LIN {X 0,Y 528.523,Z 411.8,A -85,B 0,C 180,E1 -4791.18,E2 -4791.18} C_VEL
LIN {X 0,Y 525.787,Z 397.886,A -85,B 0,C 180,E1 -4791.509,E2 -4791.509} C_VEL
LIN {X 0,Y 526.468,Z 375.264,A -85,B 0,C 180,E1 -4794.446,E2 -4794.446} C_VEL
LIN {X 0,Y 526.876,Z 362.602,A -85,B 0,C 180,E1 -4796.116,E2 -4796.116} C_VEL
LIN {X 0,Y 525.642,Z 356.23,A -85,B 0,C 180,E1 -4797.039,E2 -4797.039} C_VEL
LIN {X 0,Y 523.959,Z 348.847,A -85,B 0,C 180,E1 -4798.163,E2 -4798.163} C_VEL
LIN {X 0,Y 523.939,Z 348.847,A -85,B 0,C 180,E1 -4800.854,E2 -4800.854} C_VEL
LIN {X 0,Y 523.93,Z 348.846,A -85,B 0,C 180,E1 -4803.73,E2 -4803.73} C_VEL
LIN {X 0,Y 523.887,Z 348.853,A -85,B 0,C 180,E1 -4806.399,E2 -4806.399} C_VEL
LIN {X 0,Y 523.91,Z 348.844,A -85,B 0,C 180,E1 -4809.086,E2 -4809.086} C_VEL
LIN {X 0,Y 523.909,Z 348.848,A -85,B 0,C 180,E1 -4812.123,E2 -4812.123} C_VEL
LIN {X 0,Y 523.933,Z 348.842,A -85,B 0,C 180,E1 -4815.311,E2 -4815.311} C_VEL
LIN {X 0,Y 523.919,Z 348.849,A -85,B 0,C 180,E1 -4818.695,E2 -4818.695} C_VEL
LIN {X 0,Y 523.903,Z 348.848,A -85,B 0,C 180,E1 -4821.897,E2 -4821.897} C_VEL
LIN {X 0,Y 523.921,Z 348.844,A -85,B 0,C 180,E1 -4824.912,E2 -4824.912} C_VEL
LIN {X 0,Y 523.935,Z 348.841,A -85,B 0,C 180,E1 -4827.68,E2 -4827.68} C_VEL
LIN {X 0,Y 523.952,Z 348.844,A -85,B 0,C 180,E1 -4830.677,E2 -4830.677} C_VEL
LIN {X 0,Y 523.926,Z 348.842,A -85,B 0,C 180,E1 -4833.726,E2 -4833.726} C_VEL
LIN {X 0,Y 523.909,Z 348.852,A -85,B 0,C 180,E1 -4836.27,E2 -4836.27} C_VEL
LIN {X 0,Y 523.945,Z 348.844,A -85,B 0,C 180,E1 -4838.767,E2 -4838.767} C_VEL
LIN {X 0,Y 523.936,Z 348.841,A -85,B 0,C 180,E1 -4841.22,E2 -4841.22} C_VEL
LIN {X 0,Y 523.892,Z 348.846,A -85,B 0,C 180,E1 -4843.638,E2 -4843.638} C_VEL
LIN {X 0,Y 523.925,Z 348.846,A -85,B 0,C 180,E1 -4846.028,E2 -4846.028} C_VEL
LIN {X 0,Y 523.994,Z 348.835,A -85,B 0,C 180,E1 -4849.177,E2 -4849.177} C_VEL
LIN {X 0,Y 523.978,Z 348.84,A -85,B 0,C 180,E1 -4852.292,E2 -4852.292} C_VEL
LIN {X 0,Y 524.067,Z 348.829,A -85,B 0,C 180,E1 -4854.614,E2 -4854.614} C_VEL
LIN {X 0,Y 524.11,Z 348.82,A -85,B 0,C 180,E1 -4857.695,E2 -4857.695} C_VEL
LIN {X 0,Y 524.121,Z 348.823,A -85,B 0,C 180,E1 -4860.769,E2 -4860.769} C_VEL
LIN {X 0,Y 524.031,Z 348.828,A -85,B 0,C 180,E1 -4863.075,E2 -4863.075} C_VEL
LIN {X 0,Y 524.012,Z 348.837,A -85,B 0,C 180,E1 -4866.16,E2 -4866.16} C_VEL
LIN {X 0,Y 523.984,Z 348.836,A -85,B 0,C 180,E1 -4869.263,E2 -4869.263} C_VEL
LIN {X 0,Y 524.002,Z 348.832,A -85,B 0,C 180,E1 -4871.737,E2 -4871.737} C_VEL
LIN {X 0,Y 523.997,Z 348.835,A -85,B 0,C 180,E1 -4875.053,E2 -4875.053} C_VEL
LIN {X 0,Y 523.948,Z 348.841,A -85,B 0,C 180,E1 -4877.97,E2 -4877.97} C_VEL
LIN {X 0,Y 523.975,Z 348.835,A -85,B 0,C 180,E1 -4880.41,E2 -4880.41} C_VEL
LIN {X 0,Y 523.913,Z 348.848,A -85,B 0,C 180,E1 -4882.894,E2 -4882.894} C_VEL
LIN {X 0,Y 523.905,Z 348.838,A -85,B 0,C 180,E1 -4885.422,E2 -4885.422} C_VEL
LIN {X 0,Y 523.917,Z 348.845,A -85,B 0,C 180,E1 -4888.002,E2 -4888.002} C_VEL
LIN {X 0,Y 523.948,Z 348.84,A -85,B 0,C 180,E1 -4890.855,E2 -4890.855} C_VEL
LIN {X 0,Y 523.933,Z 348.843,A -85,B 0,C 180,E1 -4893.73,E2 -4893.73} C_VEL
LIN {X 0,Y 523.892,Z 348.849,A -85,B 0,C 180,E1 -4896.399,E2 -4896.399} C_VEL
LIN {X 0,Y 523.915,Z 348.843,A -85,B 0,C 180,E1 -4899.086,E2 -4899.086} C_VEL
LIN {X 0,Y 523.914,Z 348.848,A -85,B 0,C 180,E1 -4902.123,E2 -4902.123} C_VEL
LIN {X 0,Y 523.944,Z 348.84,A -85,B 0,C 180,E1 -4905.311,E2 -4905.311} C_VEL
LIN {X 0,Y 523.904,Z 348.849,A -85,B 0,C 180,E1 -4906.909,E2 -4906.909} C_VEL
LIN {X 0,Y 523.24,Z 348.929,A -85,B 0,C 180,E1 -4907.551,E2 -4907.551} C_VEL
LIN {X 0,Y 520.398,Z 349.291,A -85,B 0,C 180,E1 -4908.593,E2 -4908.593} C_VEL
LIN {X 0,Y 517.994,Z 349.592,A -85,B 0,C 180,E1 -4909.432,E2 -4909.432} C_VEL
LIN {X 0,Y 516.961,Z 349.719,A -85,B 0,C 180,E1 -4910.08,E2 -4910.08} C_VEL
LIN {X 0,Y 516.877,Z 349.728,A -85,B 0,C 180,E1 -4910.299,E2 -4910.299} C_VEL
LIN {X 0,Y 516.857,Z 349.726,A -85,B 0,C 180,E1 -4913.347,E2 -4913.347} C_VEL
LIN {X 0,Y 516.896,Z 349.753,A -85,B 0,C 180,E1 -4915.084,E2 -4915.084} C_VEL
LIN {X 0,Y 519.011,Z 359.38,A -85,B 0,C 180,E1 -4916.734,E2 -4916.734} C_VEL
LIN {X 0,Y 518.863,Z 369.351,A -85,B 0,C 180,E1 -4918.268,E2 -4918.268} C_VEL
LIN {X 0,Y 521.979,Z 382.993,A -85,B 0,C 180,E1 -4918.604,E2 -4918.604} C_VEL
LIN {X 0,Y 520.819,Z 533.898,A -85,B 0,C 180,E1 -4920.756,E2 -4920.756} C_VEL
LIN {X 0,Y 520.565,Z 549.845,A -85,B 0,C 180,E1 -4921.151,E2 -4921.151} C_VEL
LIN {X 0,Y 520.145,Z 564.573,A -85,B 0,C 180,E1 -4921.675,E2 -4921.675} C_VEL
LIN {X 0,Y 519.695,Z 577.889,A -85,B 0,C 180,E1 -4922.299,E2 -4922.299} C_VEL
LIN {X 0,Y 519.253,Z 591.998,A -85,B 0,C 180,E1 -4923.131,E2 -4923.131} C_VEL
LIN {X 0,Y 518.677,Z 605.217,A -85,B 0,C 180,E1 -4924.088,E2 -4924.088} C_VEL
LIN {X 0,Y 518.211,Z 617.164,A -85,B 0,C 180,E1 -4925.139,E2 -4925.139} C_VEL
LIN {X 0,Y 517.773,Z 627.214,A -85,B 0,C 180,E1 -4926.183,E2 -4926.183} C_VEL
LIN {X 0,Y 517.288,Z 637.933,A -85,B 0,C 180,E1 -4927.499,E2 -4927.499} C_VEL
LIN {X 0,Y 516.945,Z 647.314,A -85,B 0,C 180,E1 -4928.883,E2 -4928.883} C_VEL
LIN {X 0,Y 516.665,Z 655.438,A -85,B 0,C 180,E1 -4930.326,E2 -4930.326} C_VEL
LIN {X 0,Y 516.495,Z 662.099,A -85,B 0,C 180,E1 -4931.762,E2 -4931.762} C_VEL
LIN {X 0,Y 516.351,Z 668.133,A -85,B 0,C 180,E1 -4933.392,E2 -4933.392} C_VEL
LIN {X 0,Y 516.309,Z 672.687,A -85,B 0,C 180,E1 -4935.011,E2 -4935.011} C_VEL
LIN {X 0,Y 516.185,Z 675.904,A -85,B 0,C 180,E1 -4936.617,E2 -4936.617} C_VEL
LIN {X 0,Y 516.231,Z 677.854,A -85,B 0,C 180,E1 -4938.217,E2 -4938.217} C_VEL
LIN {X 0,Y 516.221,Z 678.594,A -85,B 0,C 180,E1 -4939.806,E2 -4939.806} C_VEL
LIN {X 0,Y 516.195,Z 678.184,A -85,B 0,C 180,E1 -4941.387,E2 -4941.387} C_VEL
LIN {X 0,Y 516.284,Z 676.629,A -85,B 0,C 180,E1 -4942.963,E2 -4942.963} C_VEL
LIN {X 0,Y 516.313,Z 673.92,A -85,B 0,C 180,E1 -4944.532,E2 -4944.532} C_VEL
LIN {X 0,Y 516.387,Z 669.998,A -85,B 0,C 180,E1 -4946.098,E2 -4946.098} C_VEL
LIN {X 0,Y 516.37,Z 664.776,A -85,B 0,C 180,E1 -4947.66,E2 -4947.66} C_VEL
LIN {X 0,Y 516.574,Z 658.136,A -85,B 0,C 180,E1 -4949.221,E2 -4949.221} C_VEL
LIN {X 0,Y 516.805,Z 651.008,A -85,B 0,C 180,E1 -4950.584,E2 -4950.584} C_VEL
LIN {X 0,Y 517.127,Z 642.494,A -85,B 0,C 180,E1 -4951.947,E2 -4951.947} C_VEL
LIN {X 0,Y 517.55,Z 632.309,A -85,B 0,C 180,E1 -4953.309,E2 -4953.309} C_VEL
LIN {X 0,Y 517.995,Z 621.915,A -85,B 0,C 180,E1 -4954.474,E2 -4954.474} C_VEL
LIN {X 0,Y 518.569,Z 609.495,A -85,B 0,C 180,E1 -4955.639,E2 -4955.639} C_VEL
LIN {X 0,Y 519.043,Z 597.067,A -85,B 0,C 180,E1 -4956.609,E2 -4956.609} C_VEL
LIN {X 0,Y 519.514,Z 585.147,A -85,B 0,C 180,E1 -4957.384,E2 -4957.384} C_VEL
LIN {X 0,Y 519.995,Z 570.33,A -85,B 0,C 180,E1 -4958.159,E2 -4958.159} C_VEL
LIN {X 0,Y 520.421,Z 555.2,A -85,B 0,C 180,E1 -4958.763,E2 -4958.763} C_VEL
LIN {X 0,Y 520.754,Z 540.07,A -85,B 0,C 180,E1 -4959.198,E2 -4959.198} C_VEL
LIN {X 0,Y 520.967,Z 524.806,A -85,B 0,C 180,E1 -4959.479,E2 -4959.479} C_VEL
LIN {X 0,Y 521.921,Z 382.993,A -85,B 0,C 180,E1 -4961.486,E2 -4961.486} C_VEL
LIN {X 0,Y 518.805,Z 368.955,A -85,B 0,C 180,E1 -4961.848,E2 -4961.848} C_VEL
LIN {X 0,Y 518.989,Z 359.611,A -85,B 0,C 180,E1 -4963.309,E2 -4963.309} C_VEL
LIN {X 0,Y 516.945,Z 349.72,A -85,B 0,C 180,E1 -4965.021,E2 -4965.021} C_VEL
LIN {X 0,Y 516.884,Z 349.724,A -85,B 0,C 180,E1 -4968.224,E2 -4968.224} C_VEL
LIN {X 0,Y 516.91,Z 349.717,A -85,B 0,C 180,E1 -4970.702,E2 -4970.702} C_VEL
LIN {X 0,Y 516.89,Z 349.722,A -85,B 0,C 180,E1 -4974.073,E2 -4974.073} C_VEL
LIN {X 0,Y 516.849,Z 349.725,A -85,B 0,C 180,E1 -4976.662,E2 -4976.662} C_VEL
LIN {X 0,Y 516.891,Z 349.725,A -85,B 0,C 180,E1 -4979.519,E2 -4979.519} C_VEL
LIN {X 0,Y 516.9,Z 349.715,A -85,B 0,C 180,E1 -4982.543,E2 -4982.543} C_VEL
LIN {X 0,Y 516.858,Z 349.729,A -85,B 0,C 180,E1 -4985.327,E2 -4985.327} C_VEL
LIN {X 0,Y 516.88,Z 349.721,A -85,B 0,C 180,E1 -4988.716,E2 -4988.716} C_VEL
LIN {X 0,Y 516.854,Z 349.729,A -85,B 0,C 180,E1 -4991.781,E2 -4991.781} C_VEL
LIN {X 0,Y 516.9,Z 349.718,A -85,B 0,C 180,E1 -4995.007,E2 -4995.007} C_VEL
LIN {X 0,Y 516.891,Z 349.719,A -85,B 0,C 180,E1 -4998.402,E2 -4998.402} C_VEL
LIN {X 0,Y 516.878,Z 349.724,A -85,B 0,C 180,E1 -5001.283,E2 -5001.283} C_VEL
LIN {X 0,Y 516.863,Z 349.722,A -85,B 0,C 180,E1 -5004.671,E2 -5004.671} C_VEL
LIN {X 0,Y 516.898,Z 349.724,A -85,B 0,C 180,E1 -5007.457,E2 -5007.457} C_VEL
LIN {X 0,Y 516.923,Z 349.713,A -85,B 0,C 180,E1 -5010.695,E2 -5010.695} C_VEL
LIN {X 0,Y 516.883,Z 349.711,A -85,B 0,C 180,E1 -5013.818,E2 -5013.818} C_VEL
LIN {X 0,Y 516.862,Z 349.719,A -85,B 0,C 180,E1 -5016.776,E2 -5016.776} C_VEL
LIN {X 0,Y 516.943,Z 349.719,A -85,B 0,C 180,E1 -5019.731,E2 -5019.731} C_VEL
LIN {X 0,Y 516.899,Z 349.713,A -85,B 0,C 180,E1 -5022.595,E2 -5022.595} C_VEL
LIN {X 0,Y 516.939,Z 349.714,A -85,B 0,C 180,E1 -5025.03,E2 -5025.03} C_VEL
LIN {X 0,Y 516.97,Z 349.704,A -85,B 0,C 180,E1 -5028.233,E2 -5028.233} C_VEL
LIN {X 0,Y 516.934,Z 349.718,A -85,B 0,C 180,E1 -5031.399,E2 -5031.399} C_VEL
LIN {X 0,Y 516.99,Z 349.702,A -85,B 0,C 180,E1 -5034.539,E2 -5034.539} C_VEL
LIN {X 0,Y 517.078,Z 349.704,A -85,B 0,C 180,E1 -5037.663,E2 -5037.663} C_VEL
LIN {X 0,Y 517.071,Z 349.697,A -85,B 0,C 180,E1 -5040,E2 -5040} C_VEL
LIN {X 0,Y 517.081,Z 349.693,A -85,B 0,C 180,E1 -5042.337,E2 -5042.337} C_VEL
LIN {X 0,Y 516.978,Z 349.708,A -85,B 0,C 180,E1 -5046.243,E2 -5046.243} C_VEL
LIN {X 0,Y 516.939,Z 349.716,A -85,B 0,C 180,E1 -5049.389,E2 -5049.389} C_VEL
LIN {X 0,Y 516.955,Z 349.714,A -85,B 0,C 180,E1 -5051.806,E2 -5051.806} C_VEL
LIN {X 0,Y 516.941,Z 349.714,A -85,B 0,C 180,E1 -5055.143,E2 -5055.143} C_VEL
LIN {X 0,Y 516.878,Z 349.719,A -85,B 0,C 180,E1 -5058.224,E2 -5058.224} C_VEL
LIN {X 0,Y 516.906,Z 349.716,A -85,B 0,C 180,E1 -5060.701,E2 -5060.701} C_VEL
LIN {X 0,Y 516.886,Z 349.722,A -85,B 0,C 180,E1 -5064.073,E2 -5064.073} C_VEL
LIN {X 0,Y 516.851,Z 349.722,A -85,B 0,C 180,E1 -5066.662,E2 -5066.662} C_VEL
LIN {X 0,Y 516.887,Z 349.727,A -85,B 0,C 180,E1 -5069.518,E2 -5069.518} C_VEL
LIN {X 0,Y 516.896,Z 349.718,A -85,B 0,C 180,E1 -5072.543,E2 -5072.543} C_VEL
LIN {X 0,Y 516.853,Z 349.728,A -85,B 0,C 180,E1 -5075.327,E2 -5075.327} C_VEL
LIN {X 0,Y 516.874,Z 349.719,A -85,B 0,C 180,E1 -5078.716,E2 -5078.716} C_VEL
LIN {X 0,Y 516.85,Z 349.731,A -85,B 0,C 180,E1 -5081.781,E2 -5081.781} C_VEL
LIN {X 0,Y 516.895,Z 349.72,A -85,B 0,C 180,E1 -5085.007,E2 -5085.007} C_VEL
LIN {X 0,Y 516.887,Z 349.721,A -85,B 0,C 180,E1 -5088.402,E2 -5088.402} C_VEL
LIN {X 0,Y 516.873,Z 349.727,A -85,B 0,C 180,E1 -5091.283,E2 -5091.283} C_VEL
LIN {X 0,Y 516.86,Z 349.724,A -85,B 0,C 180,E1 -5094.671,E2 -5094.671} C_VEL
LIN {X 0,Y 516.894,Z 349.726,A -85,B 0,C 180,E1 -5097.457,E2 -5097.457} C_VEL
LIN {X 0,Y 516.92,Z 349.719,A -85,B 0,C 180,E1 -5100.695,E2 -5100.695} C_VEL
LIN {X 0,Y 516.897,Z 349.847,A -85,B 0,C 180,E1 -5101.606,E2 -5101.606} C_VEL
LIN {X 0,Y 519.884,Z 362.48,A -85,B 0,C 180,E1 -5103.506,E2 -5103.506} C_VEL
LIN {X 0,Y 519.893,Z 370.17,A -85,B 0,C 180,E1 -5104.553,E2 -5104.553} C_VEL
LIN {X 0,Y 519.119,Z 391.367,A -85,B 0,C 180,E1 -5107.36,E2 -5107.36} C_VEL
LIN {X 0,Y 518.927,Z 397.801,A -85,B 0,C 180,E1 -5108.203,E2 -5108.203} C_VEL
LIN {X 0,Y 521.926,Z 413.084,A -85,B 0,C 180,E1 -5108.56,E2 -5108.56} C_VEL
LIN {X 0,Y 520.871,Z 563.853,A -85,B 0,C 180,E1 -5110.706,E2 -5110.706} C_VEL
LIN {X 0,Y 520.509,Z 578.962,A -85,B 0,C 180,E1 -5111.066,E2 -5111.066} C_VEL
LIN {X 0,Y 520.139,Z 593.99,A -85,B 0,C 180,E1 -5111.588,E2 -5111.588} C_VEL
LIN {X 0,Y 519.659,Z 607.046,A -85,B 0,C 180,E1 -5112.182,E2 -5112.182} C_VEL
LIN {X 0,Y 519.18,Z 620.988,A -85,B 0,C 180,E1 -5112.978,E2 -5112.978} C_VEL
LIN {X 0,Y 518.647,Z 634.277,A -85,B 0,C 180,E1 -5113.912,E2 -5113.912} C_VEL
LIN {X 0,Y 518.182,Z 645.793,A -85,B 0,C 180,E1 -5114.884,E2 -5114.884} C_VEL
LIN {X 0,Y 517.683,Z 657.488,A -85,B 0,C 180,E1 -5116.056,E2 -5116.056} C_VEL
LIN {X 0,Y 517.304,Z 667.496,A -85,B 0,C 180,E1 -5117.246,E2 -5117.246} C_VEL
LIN {X 0,Y 516.945,Z 677.288,A -85,B 0,C 180,E1 -5118.631,E2 -5118.631} C_VEL
LIN {X 0,Y 516.677,Z 685.457,A -85,B 0,C 180,E1 -5120.013,E2 -5120.013} C_VEL
LIN {X 0,Y 516.54,Z 692.211,A -85,B 0,C 180,E1 -5121.392,E2 -5121.392} C_VEL
LIN {X 0,Y 516.391,Z 698.449,A -85,B 0,C 180,E1 -5122.964,E2 -5122.964} C_VEL
LIN {X 0,Y 516.352,Z 703.276,A -85,B 0,C 180,E1 -5124.533,E2 -5124.533} C_VEL
LIN {X 0,Y 516.307,Z 706.811,A -85,B 0,C 180,E1 -5126.097,E2 -5126.097} C_VEL
LIN {X 0,Y 516.258,Z 709.136,A -85,B 0,C 180,E1 -5127.659,E2 -5127.659} C_VEL
LIN {X 0,Y 516.156,Z 710.303,A -85,B 0,C 180,E1 -5129.22,E2 -5129.22} C_VEL
LIN {X 0,Y 516.156,Z 710.302,A -85,B 0,C 180,E1 -5130.78,E2 -5130.78} C_VEL
LIN {X 0,Y 516.258,Z 709.131,A -85,B 0,C 180,E1 -5132.341,E2 -5132.341} C_VEL
LIN {X 0,Y 516.307,Z 706.806,A -85,B 0,C 180,E1 -5133.903,E2 -5133.903} C_VEL
LIN {X 0,Y 516.351,Z 703.276,A -85,B 0,C 180,E1 -5135.467,E2 -5135.467} C_VEL
LIN {X 0,Y 516.391,Z 698.45,A -85,B 0,C 180,E1 -5137.036,E2 -5137.036} C_VEL
LIN {X 0,Y 516.54,Z 692.202,A -85,B 0,C 180,E1 -5138.607,E2 -5138.607} C_VEL
LIN {X 0,Y 516.757,Z 684.355,A -85,B 0,C 180,E1 -5140.184,E2 -5140.184} C_VEL
LIN {X 0,Y 516.998,Z 676.009,A -85,B 0,C 180,E1 -5141.567,E2 -5141.567} C_VEL
LIN {X 0,Y 517.383,Z 665.957,A -85,B 0,C 180,E1 -5142.952,E2 -5142.952} C_VEL
LIN {X 0,Y 517.747,Z 655.676,A -85,B 0,C 180,E1 -5144.143,E2 -5144.143} C_VEL
LIN {X 0,Y 518.27,Z 643.713,A -85,B 0,C 180,E1 -5145.307,E2 -5145.307} C_VEL
LIN {X 0,Y 518.781,Z 631.145,A -85,B 0,C 180,E1 -5146.326,E2 -5146.326} C_VEL
LIN {X 0,Y 519.326,Z 617.773,A -85,B 0,C 180,E1 -5147.219,E2 -5147.219} C_VEL
LIN {X 0,Y 519.754,Z 605.012,A -85,B 0,C 180,E1 -5147.916,E2 -5147.916} C_VEL
LIN {X 0,Y 520.215,Z 590.051,A -85,B 0,C 180,E1 -5148.562,E2 -5148.562} C_VEL
LIN {X 0,Y 520.547,Z 575.06,A -85,B 0,C 180,E1 -5149.04,E2 -5149.04} C_VEL
LIN {X 0,Y 520.87,Z 559.843,A -85,B 0,C 180,E1 -5149.361,E2 -5149.361} C_VEL
LIN {X 0,Y 521.868,Z 412.692,A -85,B 0,C 180,E1 -5151.448,E2 -5151.448} C_VEL
LIN {X 0,Y 518.907,Z 397.728,A -85,B 0,C 180,E1 -5151.799,E2 -5151.799} C_VEL
LIN {X 0,Y 519.609,Z 376.635,A -85,B 0,C 180,E1 -5154.577,E2 -5154.577} C_VEL
LIN {X 0,Y 520.03,Z 363.985,A -85,B 0,C 180,E1 -5156.27,E2 -5156.27} C_VEL
LIN {X 0,Y 517.499,Z 352.265,A -85,B 0,C 180,E1 -5158.025,E2 -5158.025} C_VEL
LIN {X 0,Y 516.903,Z 349.726,A -85,B 0,C 180,E1 -5158.416,E2 -5158.416} C_VEL
LIN {X 0,Y 516.887,Z 349.724,A -85,B 0,C 180,E1 -5161.11,E2 -5161.11} C_VEL
LIN {X 0,Y 516.885,Z 349.726,A -85,B 0,C 180,E1 -5163.962,E2 -5163.962} C_VEL
LIN {X 0,Y 516.843,Z 349.73,A -85,B 0,C 180,E1 -5166.749,E2 -5166.749} C_VEL
LIN {X 0,Y 516.857,Z 349.723,A -85,B 0,C 180,E1 -5169.724,E2 -5169.724} C_VEL
LIN {X 0,Y 516.883,Z 349.72,A -85,B 0,C 180,E1 -5171.778,E2 -5171.778} C_VEL
LIN {X 0,Y 516.895,Z 349.721,A -85,B 0,C 180,E1 -5175.007,E2 -5175.007} C_VEL
LIN {X 0,Y 516.855,Z 349.731,A -85,B 0,C 180,E1 -5178.406,E2 -5178.406} C_VEL
LIN {X 0,Y 516.873,Z 349.722,A -85,B 0,C 180,E1 -5181.284,E2 -5181.284} C_VEL
LIN {X 0,Y 516.862,Z 349.726,A -85,B 0,C 180,E1 -5184.671,E2 -5184.671} C_VEL
LIN {X 0,Y 516.896,Z 349.717,A -85,B 0,C 180,E1 -5187.457,E2 -5187.457} C_VEL
LIN {X 0,Y 516.919,Z 349.72,A -85,B 0,C 180,E1 -5190.696,E2 -5190.696} C_VEL
LIN {X 0,Y 516.894,Z 349.719,A -85,B 0,C 180,E1 -5193.815,E2 -5193.815} C_VEL
LIN {X 0,Y 516.858,Z 349.726,A -85,B 0,C 180,E1 -5196.776,E2 -5196.776} C_VEL
LIN {X 0,Y 516.938,Z 349.714,A -85,B 0,C 180,E1 -5199.733,E2 -5199.733} C_VEL
LIN {X 0,Y 516.885,Z 349.725,A -85,B 0,C 180,E1 -5202.595,E2 -5202.595} C_VEL
LIN {X 0,Y 516.936,Z 349.715,A -85,B 0,C 180,E1 -5205.03,E2 -5205.03} C_VEL
LIN {X 0,Y 516.968,Z 349.713,A -85,B 0,C 180,E1 -5208.234,E2 -5208.234} C_VEL
LIN {X 0,Y 516.954,Z 349.709,A -85,B 0,C 180,E1 -5211.4,E2 -5211.4} C_VEL
LIN {X 0,Y 517.013,Z 349.709,A -85,B 0,C 180,E1 -5214.54,E2 -5214.54} C_VEL
LIN {X 0,Y 517.081,Z 349.696,A -85,B 0,C 180,E1 -5217.663,E2 -5217.663} C_VEL
LIN {X 0,Y 517.091,Z 349.699,A -85,B 0,C 180,E1 -5220.779,E2 -5220.779} C_VEL
LIN {X 0,Y 516.973,Z 349.707,A -85,B 0,C 180,E1 -5223.118,E2 -5223.118} C_VEL
LIN {X 0,Y 516.977,Z 349.714,A -85,B 0,C 180,E1 -5226.244,E2 -5226.244} C_VEL
LIN {X 0,Y 516.94,Z 349.713,A -85,B 0,C 180,E1 -5229.39,E2 -5229.39} C_VEL
LIN {X 0,Y 516.955,Z 349.71,A -85,B 0,C 180,E1 -5231.807,E2 -5231.807} C_VEL
LIN {X 0,Y 516.948,Z 349.712,A -85,B 0,C 180,E1 -5235.147,E2 -5235.147} C_VEL
LIN {X 0,Y 516.916,Z 349.72,A -85,B 0,C 180,E1 -5238.223,E2 -5238.223} C_VEL
LIN {X 0,Y 516.916,Z 349.718,A -85,B 0,C 180,E1 -5240.702,E2 -5240.702} C_VEL
LIN {X 0,Y 516.889,Z 349.722,A -85,B 0,C 180,E1 -5244.074,E2 -5244.074} C_VEL
LIN {X 0,Y 516.844,Z 349.727,A -85,B 0,C 180,E1 -5246.663,E2 -5246.663} C_VEL
LIN {X 0,Y 516.913,Z 349.715,A -85,B 0,C 180,E1 -5249.524,E2 -5249.524} C_VEL
LIN {X 0,Y 516.898,Z 349.724,A -85,B 0,C 180,E1 -5252.543,E2 -5252.543} C_VEL
LIN {X 0,Y 516.865,Z 349.717,A -85,B 0,C 180,E1 -5255.329,E2 -5255.329} C_VEL
LIN {X 0,Y 516.878,Z 349.723,A -85,B 0,C 180,E1 -5258.717,E2 -5258.717} C_VEL
LIN {X 0,Y 516.888,Z 349.721,A -85,B 0,C 180,E1 -5261.778,E2 -5261.778} C_VEL
LIN {X 0,Y 516.899,Z 349.72,A -85,B 0,C 180,E1 -5265.007,E2 -5265.007} C_VEL
LIN {X 0,Y 516.907,Z 349.723,A -85,B 0,C 180,E1 -5268.4,E2 -5268.4} C_VEL
LIN {X 0,Y 516.877,Z 349.728,A -85,B 0,C 180,E1 -5270.299,E2 -5270.299} C_VEL
LIN {X 0,Y 516.208,Z 349.81,A -85,B 0,C 180,E1 -5270.949,E2 -5270.949} C_VEL
LIN {X 0,Y 513.354,Z 350.164,A -85,B 0,C 180,E1 -5272.005,E2 -5272.005} C_VEL
LIN {X 0,Y 510.938,Z 350.464,A -85,B 0,C 180,E1 -5272.855,E2 -5272.855} C_VEL
LIN {X 0,Y 509.897,Z 350.593,A -85,B 0,C 180,E1 -5273.512,E2 -5273.512} C_VEL
LIN {X 0,Y 509.81,Z 350.604,A -85,B 0,C 180,E1 -5273.734,E2 -5273.734} C_VEL
LIN {X 0,Y 509.891,Z 350.741,A -85,B 0,C 180,E1 -5274.838,E2 -5274.838} C_VEL
LIN {X 0,Y 512.204,Z 361.496,A -85,B 0,C 180,E1 -5276.712,E2 -5276.712} C_VEL
LIN {X 0,Y 512.04,Z 369.598,A -85,B 0,C 180,E1 -5277.963,E2 -5277.963} C_VEL
LIN {X 0,Y 515.38,Z 384.215,A -85,B 0,C 180,E1 -5278.331,E2 -5278.331} C_VEL
LIN {X 0,Y 514.138,Z 534.651,A -85,B 0,C 180,E1 -5280.507,E2 -5280.507} C_VEL
LIN {X 0,Y 513.841,Z 550.586,A -85,B 0,C 180,E1 -5280.912,E2 -5280.912} C_VEL
LIN {X 0,Y 513.405,Z 564.857,A -85,B 0,C 180,E1 -5281.428,E2 -5281.428} C_VEL
LIN {X 0,Y 512.895,Z 579.335,A -85,B 0,C 180,E1 -5282.121,E2 -5282.121} C_VEL
LIN {X 0,Y 512.402,Z 593.563,A -85,B 0,C 180,E1 -5282.989,E2 -5282.989} C_VEL
LIN {X 0,Y 511.803,Z 606.237,A -85,B 0,C 180,E1 -5283.933,E2 -5283.933} C_VEL
LIN {X 0,Y 511.272,Z 618.323,A -85,B 0,C 180,E1 -5285.022,E2 -5285.022} C_VEL
LIN {X 0,Y 510.729,Z 629.847,A -85,B 0,C 180,E1 -5286.265,E2 -5286.265} C_VEL
LIN {X 0,Y 510.284,Z 640.066,A -85,B 0,C 180,E1 -5287.586,E2 -5287.586} C_VEL
LIN {X 0,Y 509.927,Z 649.196,A -85,B 0,C 180,E1 -5289.002,E2 -5289.002} C_VEL
LIN {X 0,Y 509.575,Z 657.01,A -85,B 0,C 180,E1 -5290.461,E2 -5290.461} C_VEL
LIN {X 0,Y 509.412,Z 664.406,A -85,B 0,C 180,E1 -5292.167,E2 -5292.167} C_VEL
LIN {X 0,Y 509.267,Z 669.18,A -85,B 0,C 180,E1 -5293.566,E2 -5293.566} C_VEL
LIN {X 0,Y 509.225,Z 673.127,A -85,B 0,C 180,E1 -5295.04,E2 -5295.04} C_VEL
LIN {X 0,Y 509.1,Z 675.892,A -85,B 0,C 180,E1 -5296.427,E2 -5296.427} C_VEL
LIN {X 0,Y 509.135,Z 677.932,A -85,B 0,C 180,E1 -5298.05,E2 -5298.05} C_VEL
LIN {X 0,Y 509.125,Z 678.785,A -85,B 0,C 180,E1 -5299.662,E2 -5299.662} C_VEL
LIN {X 0,Y 509.104,Z 678.485,A -85,B 0,C 180,E1 -5301.266,E2 -5301.266} C_VEL
LIN {X 0,Y 509.198,Z 677.042,A -85,B 0,C 180,E1 -5302.864,E2 -5302.864} C_VEL
LIN {X 0,Y 509.243,Z 674.44,A -85,B 0,C 180,E1 -5304.456,E2 -5304.456} C_VEL
LIN {X 0,Y 509.311,Z 670.591,A -85,B 0,C 180,E1 -5306.044,E2 -5306.044} C_VEL
LIN {X 0,Y 509.295,Z 665.482,A -85,B 0,C 180,E1 -5307.627,E2 -5307.627} C_VEL
LIN {X 0,Y 509.504,Z 658.974,A -85,B 0,C 180,E1 -5309.21,E2 -5309.21} C_VEL
LIN {X 0,Y 509.755,Z 651.989,A -85,B 0,C 180,E1 -5310.593,E2 -5310.593} C_VEL
LIN {X 0,Y 510.099,Z 643.635,A -85,B 0,C 180,E1 -5311.974,E2 -5311.974} C_VEL
LIN {X 0,Y 510.568,Z 633.63,A -85,B 0,C 180,E1 -5313.354,E2 -5313.354} C_VEL
LIN {X 0,Y 511.017,Z 623.459,A -85,B 0,C 180,E1 -5314.536,E2 -5314.536} C_VEL
LIN {X 0,Y 511.63,Z 611.302,A -85,B 0,C 180,E1 -5315.716,E2 -5315.716} C_VEL
LIN {X 0,Y 512.143,Z 599.208,A -85,B 0,C 180,E1 -5316.698,E2 -5316.698} C_VEL
LIN {X 0,Y 512.705,Z 586.024,A -85,B 0,C 180,E1 -5317.582,E2 -5317.582} C_VEL
LIN {X 0,Y 513.227,Z 571.393,A -85,B 0,C 180,E1 -5318.366,E2 -5318.366} C_VEL
LIN {X 0,Y 513.647,Z 557.269,A -85,B 0,C 180,E1 -5318.954,E2 -5318.954} C_VEL
LIN {X 0,Y 514.083,Z 541.909,A -85,B 0,C 180,E1 -5319.417,E2 -5319.417} C_VEL
LIN {X 0,Y 514.255,Z 527.36,A -85,B 0,C 180,E1 -5319.706,E2 -5319.706} C_VEL
LIN {X 0,Y 515.332,Z 384.044,A -85,B 0,C 180,E1 -5321.762,E2 -5321.762} C_VEL
LIN {X 0,Y 511.944,Z 369.306,A -85,B 0,C 180,E1 -5322.135,E2 -5322.135} C_VEL
LIN {X 0,Y 512.219,Z 362.031,A -85,B 0,C 180,E1 -5323.278,E2 -5323.278} C_VEL
LIN {X 0,Y 510.246,Z 352.192,A -85,B 0,C 180,E1 -5324.967,E2 -5324.967} C_VEL
LIN {X 0,Y 509.908,Z 350.596,A -85,B 0,C 180,E1 -5325.264,E2 -5325.264} C_VEL
LIN {X 0,Y 509.843,Z 350.6,A -85,B 0,C 180,E1 -5328.485,E2 -5328.485} C_VEL
LIN {X 0,Y 509.852,Z 350.597,A -85,B 0,C 180,E1 -5331.002,E2 -5331.002} C_VEL
LIN {X 0,Y 509.824,Z 350.607,A -85,B 0,C 180,E1 -5333.564,E2 -5333.564} C_VEL
LIN {X 0,Y 509.823,Z 350.6,A -85,B 0,C 180,E1 -5336.357,E2 -5336.357} C_VEL
LIN {X 0,Y 509.843,Z 350.598,A -85,B 0,C 180,E1 -5338.846,E2 -5338.846} C_VEL
LIN {X 0,Y 509.824,Z 350.605,A -85,B 0,C 180,E1 -5341.59,E2 -5341.59} C_VEL
LIN {X 0,Y 509.843,Z 350.597,A -85,B 0,C 180,E1 -5344.414,E2 -5344.414} C_VEL
LIN {X 0,Y 509.788,Z 350.607,A -85,B 0,C 180,E1 -5347.344,E2 -5347.344} C_VEL
LIN {X 0,Y 509.818,Z 350.596,A -85,B 0,C 180,E1 -5350.384,E2 -5350.384} C_VEL
LIN {X 0,Y 509.81,Z 350.609,A -85,B 0,C 180,E1 -5353.573,E2 -5353.573} C_VEL
LIN {X 0,Y 509.811,Z 350.596,A -85,B 0,C 180,E1 -5356.427,E2 -5356.427} C_VEL
LIN {X 0,Y 509.816,Z 350.606,A -85,B 0,C 180,E1 -5359.306,E2 -5359.306} C_VEL
LIN {X 0,Y 509.82,Z 350.605,A -85,B 0,C 180,E1 -5361.791,E2 -5361.791} C_VEL
LIN {X 0,Y 509.827,Z 350.599,A -85,B 0,C 180,E1 -5364.621,E2 -5364.621} C_VEL
LIN {X 0,Y 509.864,Z 350.601,A -85,B 0,C 180,E1 -5367.48,E2 -5367.48} C_VEL
LIN {X 0,Y 509.862,Z 350.593,A -85,B 0,C 180,E1 -5370.274,E2 -5370.274} C_VEL
LIN {X 0,Y 509.826,Z 350.589,A -85,B 0,C 180,E1 -5372.94,E2 -5372.94} C_VEL
LIN {X 0,Y 509.838,Z 350.593,A -85,B 0,C 180,E1 -5375.572,E2 -5375.572} C_VEL
LIN {X 0,Y 509.825,Z 350.601,A -85,B 0,C 180,E1 -5378.148,E2 -5378.148} C_VEL
LIN {X 0,Y 509.86,Z 350.594,A -85,B 0,C 180,E1 -5380.681,E2 -5380.681} C_VEL
LIN {X 0,Y 509.868,Z 350.592,A -85,B 0,C 180,E1 -5383.174,E2 -5383.174} C_VEL
LIN {X 0,Y 509.857,Z 350.603,A -85,B 0,C 180,E1 -5385.633,E2 -5385.633} C_VEL
LIN {X 0,Y 509.914,Z 350.582,A -85,B 0,C 180,E1 -5388.874,E2 -5388.874} C_VEL
LIN {X 0,Y 509.88,Z 350.594,A -85,B 0,C 180,E1 -5392.077,E2 -5392.077} C_VEL
LIN {X 0,Y 509.944,Z 350.579,A -85,B 0,C 180,E1 -5394.464,E2 -5394.464} C_VEL
LIN {X 0,Y 510.046,Z 350.58,A -85,B 0,C 180,E1 -5397.631,E2 -5397.631} C_VEL
LIN {X 0,Y 510.04,Z 350.572,A -85,B 0,C 180,E1 -5400,E2 -5400} C_VEL
LIN {X 0,Y 510.051,Z 350.568,A -85,B 0,C 180,E1 -5402.369,E2 -5402.369} C_VEL
LIN {X 0,Y 509.944,Z 350.593,A -85,B 0,C 180,E1 -5405.536,E2 -5405.536} C_VEL
LIN {X 0,Y 509.903,Z 350.587,A -85,B 0,C 180,E1 -5408.72,E2 -5408.72} C_VEL
LIN {X 0,Y 509.906,Z 350.59,A -85,B 0,C 180,E1 -5411.931,E2 -5411.931} C_VEL
LIN {X 0,Y 509.897,Z 350.592,A -85,B 0,C 180,E1 -5415.241,E2 -5415.241} C_VEL
LIN {X 0,Y 509.838,Z 350.595,A -85,B 0,C 180,E1 -5418.484,E2 -5418.484} C_VEL
LIN {X 0,Y 509.848,Z 350.597,A -85,B 0,C 180,E1 -5421.002,E2 -5421.002} C_VEL
LIN {X 0,Y 509.819,Z 350.605,A -85,B 0,C 180,E1 -5423.564,E2 -5423.564} C_VEL
LIN {X 0,Y 509.84,Z 350.596,A -85,B 0,C 180,E1 -5426.361,E2 -5426.361} C_VEL
LIN {X 0,Y 509.839,Z 350.598,A -85,B 0,C 180,E1 -5428.846,E2 -5428.846} C_VEL
LIN {X 0,Y 509.82,Z 350.608,A -85,B 0,C 180,E1 -5431.59,E2 -5431.59} C_VEL
LIN {X 0,Y 509.842,Z 350.598,A -85,B 0,C 180,E1 -5434.414,E2 -5434.414} C_VEL
LIN {X 0,Y 509.783,Z 350.609,A -85,B 0,C 180,E1 -5437.343,E2 -5437.343} C_VEL
LIN {X 0,Y 509.813,Z 350.6,A -85,B 0,C 180,E1 -5440.384,E2 -5440.384} C_VEL
LIN {X 0,Y 509.805,Z 350.61,A -85,B 0,C 180,E1 -5443.573,E2 -5443.573} C_VEL
LIN {X 0,Y 509.807,Z 350.603,A -85,B 0,C 180,E1 -5446.427,E2 -5446.427} C_VEL
LIN {X 0,Y 509.812,Z 350.607,A -85,B 0,C 180,E1 -5449.306,E2 -5449.306} C_VEL
LIN {X 0,Y 509.816,Z 350.607,A -85,B 0,C 180,E1 -5451.791,E2 -5451.791} C_VEL
LIN {X 0,Y 509.824,Z 350.601,A -85,B 0,C 180,E1 -5454.621,E2 -5454.621} C_VEL
LIN {X 0,Y 509.86,Z 350.602,A -85,B 0,C 180,E1 -5457.481,E2 -5457.481} C_VEL
LIN {X 0,Y 509.858,Z 350.6,A -85,B 0,C 180,E1 -5460.274,E2 -5460.274} C_VEL
LIN {X 0,Y 509.869,Z 350.701,A -85,B 0,C 180,E1 -5461.339,E2 -5461.339} C_VEL
LIN {X 0,Y 513.202,Z 365.434,A -85,B 0,C 180,E1 -5463.572,E2 -5463.572} C_VEL
LIN {X 0,Y 512.527,Z 384.409,A -85,B 0,C 180,E1 -5466.139,E2 -5466.139} C_VEL
LIN {X 0,Y 512.1,Z 397.614,A -85,B 0,C 180,E1 -5467.902,E2 -5467.902} C_VEL
LIN {X 0,Y 515.346,Z 414.763,A -85,B 0,C 180,E1 -5468.3,E2 -5468.3} C_VEL
LIN {X 0,Y 514.151,Z 564.432,A -85,B 0,C 180,E1 -5470.46,E2 -5470.46} C_VEL
LIN {X 0,Y 513.763,Z 580.199,A -85,B 0,C 180,E1 -5470.854,E2 -5470.854} C_VEL
LIN {X 0,Y 513.335,Z 595.002,A -85,B 0,C 180,E1 -5471.387,E2 -5471.387} C_VEL
LIN {X 0,Y 512.824,Z 608.809,A -85,B 0,C 180,E1 -5472.04,E2 -5472.04} C_VEL
LIN {X 0,Y 512.27,Z 622.345,A -85,B 0,C 180,E1 -5472.844,E2 -5472.844} C_VEL
LIN {X 0,Y 511.69,Z 636.125,A -85,B 0,C 180,E1 -5473.851,E2 -5473.851} C_VEL
LIN {X 0,Y 511.106,Z 648.597,A -85,B 0,C 180,E1 -5474.957,E2 -5474.957} C_VEL
LIN {X 0,Y 510.586,Z 660.833,A -85,B 0,C 180,E1 -5476.264,E2 -5476.264} C_VEL
LIN {X 0,Y 510.096,Z 671.709,A -85,B 0,C 180,E1 -5477.669,E2 -5477.669} C_VEL
LIN {X 0,Y 509.856,Z 680.772,A -85,B 0,C 180,E1 -5479.074,E2 -5479.074} C_VEL
LIN {X 0,Y 509.52,Z 688.283,A -85,B 0,C 180,E1 -5480.472,E2 -5480.472} C_VEL
LIN {X 0,Y 509.378,Z 695.297,A -85,B 0,C 180,E1 -5482.069,E2 -5482.069} C_VEL
LIN {X 0,Y 509.264,Z 700.811,A -85,B 0,C 180,E1 -5483.661,E2 -5483.661} C_VEL
LIN {X 0,Y 509.158,Z 704.978,A -85,B 0,C 180,E1 -5485.249,E2 -5485.249} C_VEL
LIN {X 0,Y 509.188,Z 707.902,A -85,B 0,C 180,E1 -5486.835,E2 -5486.835} C_VEL
LIN {X 0,Y 509.109,Z 709.643,A -85,B 0,C 180,E1 -5488.418,E2 -5488.418} C_VEL
LIN {X 0,Y 509.062,Z 710.239,A -85,B 0,C 180,E1 -5490,E2 -5490} C_VEL
LIN {X 0,Y 509.109,Z 709.64,A -85,B 0,C 180,E1 -5491.582,E2 -5491.582} C_VEL
LIN {X 0,Y 509.188,Z 707.895,A -85,B 0,C 180,E1 -5493.165,E2 -5493.165} C_VEL
LIN {X 0,Y 509.157,Z 704.972,A -85,B 0,C 180,E1 -5494.751,E2 -5494.751} C_VEL
LIN {X 0,Y 509.237,Z 700.807,A -85,B 0,C 180,E1 -5496.339,E2 -5496.339} C_VEL
LIN {X 0,Y 509.378,Z 695.289,A -85,B 0,C 180,E1 -5497.931,E2 -5497.931} C_VEL
LIN {X 0,Y 509.52,Z 688.263,A -85,B 0,C 180,E1 -5499.527,E2 -5499.527} C_VEL
LIN {X 0,Y 509.851,Z 680.751,A -85,B 0,C 180,E1 -5500.926,E2 -5500.926} C_VEL
LIN {X 0,Y 510.144,Z 671.69,A -85,B 0,C 180,E1 -5502.33,E2 -5502.33} C_VEL
LIN {X 0,Y 510.593,Z 660.805,A -85,B 0,C 180,E1 -5503.735,E2 -5503.735} C_VEL
LIN {X 0,Y 511.111,Z 648.571,A -85,B 0,C 180,E1 -5505.043,E2 -5505.043} C_VEL
LIN {X 0,Y 511.687,Z 636.098,A -85,B 0,C 180,E1 -5506.149,E2 -5506.149} C_VEL
LIN {X 0,Y 512.211,Z 623.828,A -85,B 0,C 180,E1 -5507.055,E2 -5507.055} C_VEL
LIN {X 0,Y 512.751,Z 610.579,A -85,B 0,C 180,E1 -5507.859,E2 -5507.859} C_VEL
LIN {X 0,Y 513.31,Z 596.15,A -85,B 0,C 180,E1 -5508.559,E2 -5508.559} C_VEL
LIN {X 0,Y 513.711,Z 582.109,A -85,B 0,C 180,E1 -5509.082,E2 -5509.082} C_VEL
LIN {X 0,Y 514.058,Z 567.104,A -85,B 0,C 180,E1 -5509.481,E2 -5509.481} C_VEL
LIN {X 0,Y 514.284,Z 545.398,A -85,B 0,C 180,E1 -5509.834,E2 -5509.834} C_VEL
LIN {X 0,Y 515.248,Z 413.666,A -85,B 0,C 180,E1 -5511.719,E2 -5511.719} C_VEL
LIN {X 0,Y 512.054,Z 397.333,A -85,B 0,C 180,E1 -5512.127,E2 -5512.127} C_VEL
LIN {X 0,Y 512.903,Z 374.855,A -85,B 0,C 180,E1 -5515.136,E2 -5515.136} C_VEL
LIN {X 0,Y 513.183,Z 365.393,A -85,B 0,C 180,E1 -5516.429,E2 -5516.429} C_VEL
LIN {X 0,Y 509.854,Z 350.603,A -85,B 0,C 180,E1 -5518.707,E2 -5518.707} C_VEL
LIN {X 0,Y 509.818,Z 350.604,A -85,B 0,C 180,E1 -5521.59,E2 -5521.59} C_VEL
LIN {X 0,Y 509.836,Z 350.606,A -85,B 0,C 180,E1 -5524.415,E2 -5524.415} C_VEL
LIN {X 0,Y 509.793,Z 350.605,A -85,B 0,C 180,E1 -5527.343,E2 -5527.343} C_VEL
LIN {X 0,Y 509.813,Z 350.609,A -85,B 0,C 180,E1 -5530.385,E2 -5530.385} C_VEL
LIN {X 0,Y 509.795,Z 350.605,A -85,B 0,C 180,E1 -5533.059,E2 -5533.059} C_VEL
LIN {X 0,Y 509.82,Z 350.603,A -85,B 0,C 180,E1 -5535.794,E2 -5535.794} C_VEL
LIN {X 0,Y 509.806,Z 350.609,A -85,B 0,C 180,E1 -5538.57,E2 -5538.57} C_VEL
LIN {X 0,Y 509.816,Z 350.602,A -85,B 0,C 180,E1 -5541.659,E2 -5541.659} C_VEL
LIN {X 0,Y 509.825,Z 350.602,A -85,B 0,C 180,E1 -5544.622,E2 -5544.622} C_VEL
LIN {X 0,Y 509.861,Z 350.593,A -85,B 0,C 180,E1 -5547.481,E2 -5547.481} C_VEL
LIN {X 0,Y 509.858,Z 350.593,A -85,B 0,C 180,E1 -5550.274,E2 -5550.274} C_VEL
LIN {X 0,Y 509.871,Z 350.592,A -85,B 0,C 180,E1 -5553.631,E2 -5553.631} C_VEL
LIN {X 0,Y 509.819,Z 350.606,A -85,B 0,C 180,E1 -5556.436,E2 -5556.436} C_VEL
LIN {X 0,Y 509.916,Z 350.59,A -85,B 0,C 180,E1 -5559.845,E2 -5559.845} C_VEL
LIN {X 0,Y 509.847,Z 350.596,A -85,B 0,C 180,E1 -5563.174,E2 -5563.174} C_VEL
LIN {X 0,Y 509.853,Z 350.596,A -85,B 0,C 180,E1 -5565.634,E2 -5565.634} C_VEL
LIN {X 0,Y 509.913,Z 350.591,A -85,B 0,C 180,E1 -5568.875,E2 -5568.875} C_VEL
LIN {X 0,Y 509.91,Z 350.59,A -85,B 0,C 180,E1 -5572.078,E2 -5572.078} C_VEL
LIN {X 0,Y 509.964,Z 350.588,A -85,B 0,C 180,E1 -5574.464,E2 -5574.464} C_VEL
LIN {X 0,Y 510.051,Z 350.572,A -85,B 0,C 180,E1 -5577.631,E2 -5577.631} C_VEL
LIN {X 0,Y 510.041,Z 350.577,A -85,B 0,C 180,E1 -5580.79,E2 -5580.79} C_VEL
LIN {X 0,Y 509.917,Z 350.585,A -85,B 0,C 180,E1 -5583.161,E2 -5583.161} C_VEL
LIN {X 0,Y 509.925,Z 350.594,A -85,B 0,C 180,E1 -5586.331,E2 -5586.331} C_VEL
LIN {X 0,Y 509.88,Z 350.593,A -85,B 0,C 180,E1 -5589.521,E2 -5589.521} C_VEL
LIN {X 0,Y 509.907,Z 350.589,A -85,B 0,C 180,E1 -5591.932,E2 -5591.932} C_VEL
LIN {X 0,Y 509.898,Z 350.59,A -85,B 0,C 180,E1 -5595.242,E2 -5595.242} C_VEL
LIN {X 0,Y 509.86,Z 350.595,A -85,B 0,C 180,E1 -5598.484,E2 -5598.484} C_VEL
LIN {X 0,Y 509.853,Z 350.596,A -85,B 0,C 180,E1 -5601.002,E2 -5601.002} C_VEL
LIN {X 0,Y 509.823,Z 350.599,A -85,B 0,C 180,E1 -5603.564,E2 -5603.564} C_VEL
LIN {X 0,Y 509.819,Z 350.597,A -85,B 0,C 180,E1 -5606.357,E2 -5606.357} C_VEL
LIN {X 0,Y 509.853,Z 350.599,A -85,B 0,C 180,E1 -5608.846,E2 -5608.846} C_VEL
LIN {X 0,Y 509.823,Z 350.595,A -85,B 0,C 180,E1 -5611.59,E2 -5611.59} C_VEL
LIN {X 0,Y 509.84,Z 350.603,A -85,B 0,C 180,E1 -5614.415,E2 -5614.415} C_VEL
LIN {X 0,Y 509.798,Z 350.604,A -85,B 0,C 180,E1 -5617.343,E2 -5617.343} C_VEL
LIN {X 0,Y 509.817,Z 350.604,A -85,B 0,C 180,E1 -5620.385,E2 -5620.385} C_VEL
LIN {X 0,Y 509.799,Z 350.606,A -85,B 0,C 180,E1 -5623.059,E2 -5623.059} C_VEL
LIN {X 0,Y 509.826,Z 350.599,A -85,B 0,C 180,E1 -5625.794,E2 -5625.794} C_VEL
LIN {X 0,Y 509.85,Z 350.604,A -85,B 0,C 180,E1 -5628.574,E2 -5628.574} C_VEL
LIN {X 0,Y 509.854,Z 350.599,A -85,B 0,C 180,E1 -5631.787,E2 -5631.787} C_VEL
LIN {X 0,Y 509.81,Z 350.604,A -85,B 0,C 180,E1 -5633.734,E2 -5633.734} C_VEL
LIN {X 0,Y 509.604,Z 350.993,A -85,B 0,C 180,E1 -5634.169,E2 -5634.169} C_VEL
LIN {X 0,Y 508.77,Z 352.734,A -85,B 0,C 180,E1 -5634.794,E2 -5634.794} C_VEL
LIN {X 0,Y 507.63,Z 355.422,A -85,B 0,C 180,E1 -5635.376,E2 -5635.376} C_VEL
LIN {X 0,Y 506.118,Z 359.963,A -85,B 0,C 180,E1 -5636.126,E2 -5636.126} C_VEL
LIN {X 0,Y 505.373,Z 364.766,A -85,B 0,C 180,E1 -5636.869,E2 -5636.869} C_VEL
LIN {X 0,Y 505.199,Z 369.644,A -85,B 0,C 180,E1 -5637.643,E2 -5637.643} C_VEL
LIN {X 0,Y 508.842,Z 385.728,A -85,B 0,C 180,E1 -5638.057,E2 -5638.057} C_VEL
LIN {X 0,Y 507.469,Z 534.744,A -85,B 0,C 180,E1 -5640.238,E2 -5640.238} C_VEL
LIN {X 0,Y 507.158,Z 550.532,A -85,B 0,C 180,E1 -5640.641,E2 -5640.641} C_VEL
LIN {X 0,Y 506.666,Z 565.309,A -85,B 0,C 180,E1 -5641.183,E2 -5641.183} C_VEL
LIN {X 0,Y 506.174,Z 578.732,A -85,B 0,C 180,E1 -5641.831,E2 -5641.831} C_VEL
LIN {X 0,Y 505.629,Z 592.979,A -85,B 0,C 180,E1 -5642.698,E2 -5642.698} C_VEL
LIN {X 0,Y 504.983,Z 605.91,A -85,B 0,C 180,E1 -5643.665,E2 -5643.665} C_VEL
LIN {X 0,Y 504.438,Z 617.73,A -85,B 0,C 180,E1 -5644.735,E2 -5644.735} C_VEL
LIN {X 0,Y 503.87,Z 628.758,A -85,B 0,C 180,E1 -5645.922,E2 -5645.922} C_VEL
LIN {X 0,Y 503.358,Z 639.106,A -85,B 0,C 180,E1 -5647.249,E2 -5647.249} C_VEL
LIN {X 0,Y 502.922,Z 648.514,A -85,B 0,C 180,E1 -5648.695,E2 -5648.695} C_VEL
LIN {X 0,Y 502.587,Z 656.499,A -85,B 0,C 180,E1 -5650.178,E2 -5650.178} C_VEL
LIN {X 0,Y 502.366,Z 663.202,A -85,B 0,C 180,E1 -5651.695,E2 -5651.695} C_VEL
LIN {X 0,Y 502.205,Z 668.955,A -85,B 0,C 180,E1 -5653.329,E2 -5653.329} C_VEL
LIN {X 0,Y 502.138,Z 673.327,A -85,B 0,C 180,E1 -5654.96,E2 -5654.96} C_VEL
LIN {X 0,Y 502.032,Z 675.854,A -85,B 0,C 180,E1 -5656.232,E2 -5656.232} C_VEL
LIN {X 0,Y 502.037,Z 678.011,A -85,B 0,C 180,E1 -5657.879,E2 -5657.879} C_VEL
LIN {X 0,Y 502.031,Z 678.976,A -85,B 0,C 180,E1 -5659.514,E2 -5659.514} C_VEL
LIN {X 0,Y 502.024,Z 678.787,A -85,B 0,C 180,E1 -5661.142,E2 -5661.142} C_VEL
LIN {X 0,Y 502.108,Z 677.452,A -85,B 0,C 180,E1 -5662.763,E2 -5662.763} C_VEL
LIN {X 0,Y 502.153,Z 674.916,A -85,B 0,C 180,E1 -5664.378,E2 -5664.378} C_VEL
LIN {X 0,Y 502.235,Z 671.175,A -85,B 0,C 180,E1 -5665.988,E2 -5665.988} C_VEL
LIN {X 0,Y 502.222,Z 666.188,A -85,B 0,C 180,E1 -5667.594,E2 -5667.594} C_VEL
LIN {X 0,Y 502.435,Z 659.812,A -85,B 0,C 180,E1 -5669.199,E2 -5669.199} C_VEL
LIN {X 0,Y 502.73,Z 652.967,A -85,B 0,C 180,E1 -5670.601,E2 -5670.601} C_VEL
LIN {X 0,Y 503.072,Z 644.776,A -85,B 0,C 180,E1 -5672.002,E2 -5672.002} C_VEL
LIN {X 0,Y 503.581,Z 634.952,A -85,B 0,C 180,E1 -5673.4,E2 -5673.4} C_VEL
LIN {X 0,Y 504.036,Z 624.975,A -85,B 0,C 180,E1 -5674.599,E2 -5674.599} C_VEL
LIN {X 0,Y 504.688,Z 613.08,A -85,B 0,C 180,E1 -5675.794,E2 -5675.794} C_VEL
LIN {X 0,Y 505.296,Z 599.956,A -85,B 0,C 180,E1 -5676.89,E2 -5676.89} C_VEL
LIN {X 0,Y 505.902,Z 586.861,A -85,B 0,C 180,E1 -5677.785,E2 -5677.785} C_VEL
LIN {X 0,Y 506.458,Z 572.419,A -85,B 0,C 180,E1 -5678.579,E2 -5678.579} C_VEL
LIN {X 0,Y 506.955,Z 557.17,A -85,B 0,C 180,E1 -5679.224,E2 -5679.224} C_VEL
LIN {X 0,Y 507.375,Z 541.365,A -85,B 0,C 180,E1 -5679.701,E2 -5679.701} C_VEL
LIN {X 0,Y 507.619,Z 527.041,A -85,B 0,C 180,E1 -5679.982,E2 -5679.982} C_VEL
LIN {X 0,Y 508.796,Z 385.683,A -85,B 0,C 180,E1 -5682.034,E2 -5682.034} C_VEL
LIN {X 0,Y 505.116,Z 369.466,A -85,B 0,C 180,E1 -5682.454,E2 -5682.454} C_VEL
LIN {X 0,Y 505.291,Z 363.179,A -85,B 0,C 180,E1 -5683.46,E2 -5683.46} C_VEL
LIN {X 0,Y 502.836,Z 351.478,A -85,B 0,C 180,E1 -5685.504,E2 -5685.504} C_VEL
LIN {X 0,Y 502.817,Z 351.476,A -85,B 0,C 180,E1 -5688.752,E2 -5688.752} C_VEL
LIN {X 0,Y 502.787,Z 351.478,A -85,B 0,C 180,E1 -5691.311,E2 -5691.311} C_VEL
LIN {X 0,Y 502.772,Z 351.482,A -85,B 0,C 180,E1 -5693.915,E2 -5693.915} C_VEL
LIN {X 0,Y 502.789,Z 351.476,A -85,B 0,C 180,E1 -5696.571,E2 -5696.571} C_VEL
LIN {X 0,Y 502.815,Z 351.476,A -85,B 0,C 180,E1 -5699.934,E2 -5699.934} C_VEL
LIN {X 0,Y 502.835,Z 351.469,A -85,B 0,C 180,E1 -5703.031,E2 -5703.031} C_VEL
LIN {X 0,Y 502.758,Z 351.48,A -85,B 0,C 180,E1 -5705.953,E2 -5705.953} C_VEL
LIN {X 0,Y 502.79,Z 351.478,A -85,B 0,C 180,E1 -5708.977,E2 -5708.977} C_VEL
LIN {X 0,Y 502.748,Z 351.482,A -85,B 0,C 180,E1 -5712.191,E2 -5712.191} C_VEL
LIN {X 0,Y 502.79,Z 351.478,A -85,B 0,C 180,E1 -5715.47,E2 -5715.47} C_VEL
LIN {X 0,Y 502.799,Z 351.479,A -85,B 0,C 180,E1 -5717.86,E2 -5717.86} C_VEL
LIN {X 0,Y 502.787,Z 351.476,A -85,B 0,C 180,E1 -5721.022,E2 -5721.022} C_VEL
LIN {X 0,Y 502.772,Z 351.479,A -85,B 0,C 180,E1 -5724.17,E2 -5724.17} C_VEL
LIN {X 0,Y 502.807,Z 351.474,A -85,B 0,C 180,E1 -5726.998,E2 -5726.998} C_VEL
LIN {X 0,Y 502.818,Z 351.472,A -85,B 0,C 180,E1 -5730.065,E2 -5730.065} C_VEL
LIN {X 0,Y 502.787,Z 351.466,A -85,B 0,C 180,E1 -5733.429,E2 -5733.429} C_VEL
LIN {X 0,Y 502.771,Z 351.475,A -85,B 0,C 180,E1 -5736.085,E2 -5736.085} C_VEL
LIN {X 0,Y 502.787,Z 351.476,A -85,B 0,C 180,E1 -5738.689,E2 -5738.689} C_VEL
LIN {X 0,Y 502.826,Z 351.475,A -85,B 0,C 180,E1 -5741.248,E2 -5741.248} C_VEL
LIN {X 0,Y 502.852,Z 351.467,A -85,B 0,C 180,E1 -5744.6,E2 -5744.6} C_VEL
LIN {X 0,Y 502.88,Z 351.46,A -85,B 0,C 180,E1 -5748.039,E2 -5748.039} C_VEL
LIN {X 0,Y 502.853,Z 351.469,A -85,B 0,C 180,E1 -5751.156,E2 -5751.156} C_VEL
LIN {X 0,Y 502.874,Z 351.469,A -85,B 0,C 180,E1 -5753.58,E2 -5753.58} C_VEL
LIN {X 0,Y 502.84,Z 351.467,A -85,B 0,C 180,E1 -5756.795,E2 -5756.795} C_VEL
LIN {X 0,Y 502.896,Z 351.462,A -85,B 0,C 180,E1 -5758.398,E2 -5758.398} C_VEL
LIN {X 0,Y 503.009,Z 351.448,A -85,B 0,C 180,E1 -5760,E2 -5760} C_VEL
LIN {X 0,Y 503.02,Z 351.444,A -85,B 0,C 180,E1 -5762.402,E2 -5762.402} C_VEL
LIN {X 0,Y 502.901,Z 351.469,A -85,B 0,C 180,E1 -5765.614,E2 -5765.614} C_VEL
LIN {X 0,Y 502.874,Z 351.465,A -85,B 0,C 180,E1 -5768.033,E2 -5768.033} C_VEL
LIN {X 0,Y 502.878,Z 351.468,A -85,B 0,C 180,E1 -5771.283,E2 -5771.283} C_VEL
LIN {X 0,Y 502.832,Z 351.468,A -85,B 0,C 180,E1 -5774.571,E2 -5774.571} C_VEL
LIN {X 0,Y 502.811,Z 351.472,A -85,B 0,C 180,E1 -5778.109,E2 -5778.109} C_VEL
LIN {X 0,Y 502.831,Z 351.469,A -85,B 0,C 180,E1 -5780.536,E2 -5780.536} C_VEL
LIN {X 0,Y 502.787,Z 351.474,A -85,B 0,C 180,E1 -5783.04,E2 -5783.04} C_VEL
LIN {X 0,Y 502.783,Z 351.482,A -85,B 0,C 180,E1 -5785.678,E2 -5785.678} C_VEL
LIN {X 0,Y 502.775,Z 351.478,A -85,B 0,C 180,E1 -5788.376,E2 -5788.376} C_VEL
LIN {X 0,Y 502.793,Z 351.477,A -85,B 0,C 180,E1 -5791.143,E2 -5791.143} C_VEL
LIN {X 0,Y 502.798,Z 351.479,A -85,B 0,C 180,E1 -5793.994,E2 -5793.994} C_VEL
LIN {X 0,Y 502.737,Z 351.485,A -85,B 0,C 180,E1 -5797.171,E2 -5797.171} C_VEL
LIN {X 0,Y 502.77,Z 351.481,A -85,B 0,C 180,E1 -5800.017,E2 -5800.017} C_VEL
LIN {X 0,Y 502.746,Z 351.484,A -85,B 0,C 180,E1 -5803.234,E2 -5803.234} C_VEL
LIN {X 0,Y 502.779,Z 351.485,A -85,B 0,C 180,E1 -5805.66,E2 -5805.66} C_VEL
LIN {X 0,Y 502.795,Z 351.483,A -85,B 0,C 180,E1 -5807.86,E2 -5807.86} C_VEL
LIN {X 0,Y 502.783,Z 351.48,A -85,B 0,C 180,E1 -5811.022,E2 -5811.022} C_VEL
LIN {X 0,Y 502.768,Z 351.482,A -85,B 0,C 180,E1 -5814.17,E2 -5814.17} C_VEL
LIN {X 0,Y 502.83,Z 351.474,A -85,B 0,C 180,E1 -5816.994,E2 -5816.994} C_VEL
LIN {X 0,Y 502.814,Z 351.479,A -85,B 0,C 180,E1 -5820.065,E2 -5820.065} C_VEL
LIN {X 0,Y 502.859,Z 351.669,A -85,B 0,C 180,E1 -5821.087,E2 -5821.087} C_VEL
LIN {X 0,Y 506.376,Z 366.964,A -85,B 0,C 180,E1 -5823.439,E2 -5823.439} C_VEL
LIN {X 0,Y 505.595,Z 388.601,A -85,B 0,C 180,E1 -5826.397,E2 -5826.397} C_VEL
LIN {X 0,Y 505.238,Z 397.366,A -85,B 0,C 180,E1 -5827.581,E2 -5827.581} C_VEL
LIN {X 0,Y 508.707,Z 416.075,A -85,B 0,C 180,E1 -5828.025,E2 -5828.025} C_VEL
LIN {X 0,Y 507.451,Z 564.218,A -85,B 0,C 180,E1 -5830.192,E2 -5830.192} C_VEL
LIN {X 0,Y 507.02,Z 580.012,A -85,B 0,C 180,E1 -5830.591,E2 -5830.591} C_VEL
LIN {X 0,Y 506.57,Z 595.04,A -85,B 0,C 180,E1 -5831.142,E2 -5831.142} C_VEL
LIN {X 0,Y 506.034,Z 608.576,A -85,B 0,C 180,E1 -5831.791,E2 -5831.791} C_VEL
LIN {X 0,Y 505.439,Z 622.116,A -85,B 0,C 180,E1 -5832.605,E2 -5832.605} C_VEL
LIN {X 0,Y 504.814,Z 635.898,A -85,B 0,C 180,E1 -5833.625,E2 -5833.625} C_VEL
LIN {X 0,Y 504.193,Z 648.372,A -85,B 0,C 180,E1 -5834.746,E2 -5834.746} C_VEL
LIN {X 0,Y 503.684,Z 658.833,A -85,B 0,C 180,E1 -5835.866,E2 -5835.866} C_VEL
LIN {X 0,Y 503.241,Z 668.545,A -85,B 0,C 180,E1 -5837.088,E2 -5837.088} C_VEL
LIN {X 0,Y 502.838,Z 677.688,A -85,B 0,C 180,E1 -5838.447,E2 -5838.447} C_VEL
LIN {X 0,Y 502.608,Z 685.016,A -85,B 0,C 180,E1 -5839.73,E2 -5839.73} C_VEL
LIN {X 0,Y 502.388,Z 691.77,A -85,B 0,C 180,E1 -5841.148,E2 -5841.148} C_VEL
LIN {X 0,Y 502.24,Z 698.011,A -85,B 0,C 180,E1 -5842.765,E2 -5842.765} C_VEL
LIN {X 0,Y 502.181,Z 702.839,A -85,B 0,C 180,E1 -5844.378,E2 -5844.378} C_VEL
LIN {X 0,Y 502.095,Z 706.374,A -85,B 0,C 180,E1 -5845.987,E2 -5845.987} C_VEL
LIN {X 0,Y 502.088,Z 708.7,A -85,B 0,C 180,E1 -5847.593,E2 -5847.593} C_VEL
LIN {X 0,Y 501.986,Z 709.867,A -85,B 0,C 180,E1 -5849.198,E2 -5849.198} C_VEL
LIN {X 0,Y 501.986,Z 709.865,A -85,B 0,C 180,E1 -5850.802,E2 -5850.802} C_VEL
LIN {X 0,Y 502.088,Z 708.692,A -85,B 0,C 180,E1 -5852.407,E2 -5852.407} C_VEL
LIN {X 0,Y 502.095,Z 706.363,A -85,B 0,C 180,E1 -5854.013,E2 -5854.013} C_VEL
LIN {X 0,Y 502.178,Z 702.831,A -85,B 0,C 180,E1 -5855.622,E2 -5855.622} C_VEL
LIN {X 0,Y 502.24,Z 698.002,A -85,B 0,C 180,E1 -5857.235,E2 -5857.235} C_VEL
LIN {X 0,Y 502.388,Z 691.75,A -85,B 0,C 180,E1 -5858.852,E2 -5858.852} C_VEL
LIN {X 0,Y 502.65,Z 683.899,A -85,B 0,C 180,E1 -5860.473,E2 -5860.473} C_VEL
LIN {X 0,Y 502.947,Z 675.891,A -85,B 0,C 180,E1 -5861.842,E2 -5861.842} C_VEL
LIN {X 0,Y 503.393,Z 665.492,A -85,B 0,C 180,E1 -5863.318,E2 -5863.318} C_VEL
LIN {X 0,Y 503.817,Z 655.207,A -85,B 0,C 180,E1 -5864.542,E2 -5864.542} C_VEL
LIN {X 0,Y 504.492,Z 642.817,A -85,B 0,C 180,E1 -5865.776,E2 -5865.776} C_VEL
LIN {X 0,Y 505.086,Z 629.322,A -85,B 0,C 180,E1 -5866.886,E2 -5866.886} C_VEL
LIN {X 0,Y 505.792,Z 615.655,A -85,B 0,C 180,E1 -5867.8,E2 -5867.8} C_VEL
LIN {X 0,Y 506.327,Z 601.498,A -85,B 0,C 180,E1 -5868.565,E2 -5868.565} C_VEL
LIN {X 0,Y 506.842,Z 586.181,A -85,B 0,C 180,E1 -5869.202,E2 -5869.202} C_VEL
LIN {X 0,Y 507.286,Z 570.955,A -85,B 0,C 180,E1 -5869.657,E2 -5869.657} C_VEL
LIN {X 0,Y 507.517,Z 554.938,A -85,B 0,C 180,E1 -5869.964,E2 -5869.964} C_VEL
LIN {X 0,Y 508.713,Z 415.844,A -85,B 0,C 180,E1 -5871.977,E2 -5871.977} C_VEL
LIN {X 0,Y 505.232,Z 397.119,A -85,B 0,C 180,E1 -5872.442,E2 -5872.442} C_VEL
LIN {X 0,Y 506.108,Z 375.669,A -85,B 0,C 180,E1 -5875.361,E2 -5875.361} C_VEL
LIN {X 0,Y 506.365,Z 367.043,A -85,B 0,C 180,E1 -5876.561,E2 -5876.561} C_VEL
LIN {X 0,Y 503.107,Z 352.698,A -85,B 0,C 180,E1 -5878.812,E2 -5878.812} C_VEL
LIN {X 0,Y 502.811,Z 351.478,A -85,B 0,C 180,E1 -5879.03,E2 -5879.03} C_VEL
LIN {X 0,Y 502.782,Z 351.484,A -85,B 0,C 180,E1 -5882.085,E2 -5882.085} C_VEL
LIN {X 0,Y 502.792,Z 351.48,A -85,B 0,C 180,E1 -5884.966,E2 -5884.966} C_VEL
LIN {X 0,Y 502.763,Z 351.482,A -85,B 0,C 180,E1 -5888.482,E2 -5888.482} C_VEL
LIN {X 0,Y 502.771,Z 351.478,A -85,B 0,C 180,E1 -5891.071,E2 -5891.071} C_VEL
LIN {X 0,Y 502.752,Z 351.481,A -85,B 0,C 180,E1 -5893.372,E2 -5893.372} C_VEL
LIN {X 0,Y 502.777,Z 351.479,A -85,B 0,C 180,E1 -5895.66,E2 -5895.66} C_VEL
LIN {X 0,Y 502.764,Z 351.481,A -85,B 0,C 180,E1 -5899.013,E2 -5899.013} C_VEL
LIN {X 0,Y 502.764,Z 351.484,A -85,B 0,C 180,E1 -5902.044,E2 -5902.044} C_VEL
LIN {X 0,Y 502.796,Z 351.475,A -85,B 0,C 180,E1 -5905.034,E2 -5905.034} C_VEL
LIN {X 0,Y 502.783,Z 351.478,A -85,B 0,C 180,E1 -5907.916,E2 -5907.916} C_VEL
LIN {X 0,Y 502.812,Z 351.477,A -85,B 0,C 180,E1 -5910.712,E2 -5910.712} C_VEL
LIN {X 0,Y 502.822,Z 351.47,A -85,B 0,C 180,E1 -5913.449,E2 -5913.449} C_VEL
LIN {X 0,Y 502.768,Z 351.483,A -85,B 0,C 180,E1 -5916.085,E2 -5916.085} C_VEL
LIN {X 0,Y 502.782,Z 351.482,A -85,B 0,C 180,E1 -5918.689,E2 -5918.689} C_VEL
LIN {X 0,Y 502.812,Z 351.473,A -85,B 0,C 180,E1 -5921.248,E2 -5921.248} C_VEL
LIN {X 0,Y 502.838,Z 351.475,A -85,B 0,C 180,E1 -5924.664,E2 -5924.664} C_VEL
LIN {X 0,Y 502.878,Z 351.466,A -85,B 0,C 180,E1 -5928.04,E2 -5928.04} C_VEL
LIN {X 0,Y 502.863,Z 351.465,A -85,B 0,C 180,E1 -5931.157,E2 -5931.157} C_VEL
LIN {X 0,Y 502.918,Z 351.467,A -85,B 0,C 180,E1 -5934.387,E2 -5934.387} C_VEL
LIN {X 0,Y 503.02,Z 351.447,A -85,B 0,C 180,E1 -5937.598,E2 -5937.598} C_VEL
LIN {X 0,Y 502.992,Z 351.455,A -85,B 0,C 180,E1 -5940.801,E2 -5940.801} C_VEL
LIN {X 0,Y 503.019,Z 351.454,A -85,B 0,C 180,E1 -5942.403,E2 -5942.403} C_VEL
LIN {X 0,Y 502.919,Z 351.46,A -85,B 0,C 180,E1 -5945.614,E2 -5945.614} C_VEL
LIN {X 0,Y 502.863,Z 351.471,A -85,B 0,C 180,E1 -5948.844,E2 -5948.844} C_VEL
LIN {X 0,Y 502.848,Z 351.47,A -85,B 0,C 180,E1 -5952.102,E2 -5952.102} C_VEL
LIN {X 0,Y 502.852,Z 351.467,A -85,B 0,C 180,E1 -5955.4,E2 -5955.4} C_VEL
LIN {X 0,Y 502.826,Z 351.466,A -85,B 0,C 180,E1 -5958.752,E2 -5958.752} C_VEL
LIN {X 0,Y 502.786,Z 351.475,A -85,B 0,C 180,E1 -5961.312,E2 -5961.312} C_VEL
LIN {X 0,Y 502.772,Z 351.479,A -85,B 0,C 180,E1 -5963.915,E2 -5963.915} C_VEL
LIN {X 0,Y 502.786,Z 351.476,A -85,B 0,C 180,E1 -5966.571,E2 -5966.571} C_VEL
LIN {X 0,Y 502.816,Z 351.472,A -85,B 0,C 180,E1 -5969.289,E2 -5969.289} C_VEL
LIN {X 0,Y 502.786,Z 351.475,A -85,B 0,C 180,E1 -5972.085,E2 -5972.085} C_VEL
LIN {X 0,Y 502.796,Z 351.472,A -85,B 0,C 180,E1 -5974.967,E2 -5974.967} C_VEL
LIN {X 0,Y 502.768,Z 351.483,A -85,B 0,C 180,E1 -5978.482,E2 -5978.482} C_VEL
LIN {X 0,Y 502.775,Z 351.48,A -85,B 0,C 180,E1 -5981.071,E2 -5981.071} C_VEL
LIN {X 0,Y 502.757,Z 351.482,A -85,B 0,C 180,E1 -5983.372,E2 -5983.372} C_VEL
LIN {X 0,Y 502.783,Z 351.476,A -85,B 0,C 180,E1 -5985.66,E2 -5985.66} C_VEL
LIN {X 0,Y 502.8,Z 351.48,A -85,B 0,C 180,E1 -5988.932,E2 -5988.932} C_VEL
LIN {X 0,Y 502.794,Z 351.48,A -85,B 0,C 180,E1 -5992.046,E2 -5992.046} C_VEL
LIN {X 0,Y 502.809,Z 351.555,A -85,B 0,C 180,E1 -5994.545,E2 -5994.545} C_VEL
LIN {X 0,Y 505.317,Z 362.901,A -85,B 0,C 180,E1 -5996.563,E2 -5996.563} C_VEL
LIN {X 0,Y 505.373,Z 364.766,A -85,B 0,C 180,E1 -5996.869,E2 -5996.869} C_VEL
LIN {X 0,Y 505.19,Z 367.437,A -85,B 0,C 180,E1 -5997.184,E2 -5997.184} C_VEL
LIN {X 0,Y 504.555,Z 372.52,A -85,B 0,C 180,E1 -5997.504,E2 -5997.504} C_VEL
LIN {X 0,Y 503.729,Z 378.198,A -85,B 0,C 180,E1 -5997.682,E2 -5997.682} C_VEL
LIN {X 0,Y 502.215,Z 388.62,A -85,B 0,C 180,E1 -5997.788,E2 -5997.788} C_VEL
LIN {X 0,Y 502.192,Z 394.914,A -85,B 0,C 180,E1 -5997.884,E2 -5997.884} C_VEL
LIN {X 0,Y 500.818,Z 534.85,A -85,B 0,C 180,E1 -5999.961,E2 -5999.961} C_VEL
LIN {X 0,Y 500.438,Z 550.757,A -85,B 0,C 180,E1 -6000.371,E2 -6000.371} C_VEL
LIN {X 0,Y 499.941,Z 565.942,A -85,B 0,C 180,E1 -6000.939,E2 -6000.939} C_VEL
LIN {X 0,Y 499.382,Z 580.141,A -85,B 0,C 180,E1 -6001.642,E2 -6001.642} C_VEL
LIN {X 0,Y 498.822,Z 593.99,A -85,B 0,C 180,E1 -6002.51,E2 -6002.51} C_VEL
LIN {X 0,Y 498.103,Z 606.913,A -85,B 0,C 180,E1 -6003.499,E2 -6003.499} C_VEL
LIN {X 0,Y 497.51,Z 619.16,A -85,B 0,C 180,E1 -6004.638,E2 -6004.638} C_VEL
LIN {X 0,Y 496.813,Z 631.317,A -85,B 0,C 180,E1 -6006.002,E2 -6006.002} C_VEL
LIN {X 0,Y 496.344,Z 640.555,A -85,B 0,C 180,E1 -6007.238,E2 -6007.238} C_VEL
LIN {X 0,Y 495.873,Z 650.376,A -85,B 0,C 180,E1 -6008.813,E2 -6008.813} C_VEL
LIN {X 0,Y 495.441,Z 659.03,A -85,B 0,C 180,E1 -6010.527,E2 -6010.527} C_VEL
LIN {X 0,Y 495.289,Z 664.833,A -85,B 0,C 180,E1 -6011.938,E2 -6011.938} C_VEL
LIN {X 0,Y 495.134,Z 670.002,A -85,B 0,C 180,E1 -6013.508,E2 -6013.508} C_VEL
LIN {X 0,Y 495.049,Z 674.213,A -85,B 0,C 180,E1 -6015.195,E2 -6015.195} C_VEL
LIN {X 0,Y 494.93,Z 677.106,A -85,B 0,C 180,E1 -6016.868,E2 -6016.868} C_VEL
LIN {X 0,Y 494.992,Z 678.773,A -85,B 0,C 180,E1 -6018.535,E2 -6018.535} C_VEL
LIN {X 0,Y 494.917,Z 679.271,A -85,B 0,C 180,E1 -6020.189,E2 -6020.189} C_VEL
LIN {X 0,Y 494.945,Z 678.607,A -85,B 0,C 180,E1 -6021.837,E2 -6021.837} C_VEL
LIN {X 0,Y 495.068,Z 676.607,A -85,B 0,C 180,E1 -6023.581,E2 -6023.581} C_VEL
LIN {X 0,Y 495.007,Z 673.732,A -85,B 0,C 180,E1 -6025.113,E2 -6025.113} C_VEL
LIN {X 0,Y 495.204,Z 669.484,A -85,B 0,C 180,E1 -6026.746,E2 -6026.746} C_VEL
LIN {X 0,Y 495.223,Z 663.955,A -85,B 0,C 180,E1 -6028.374,E2 -6028.374} C_VEL
LIN {X 0,Y 495.61,Z 656.949,A -85,B 0,C 180,E1 -6030,E2 -6030} C_VEL
LIN {X 0,Y 495.894,Z 649.508,A -85,B 0,C 180,E1 -6031.421,E2 -6031.421} C_VEL
LIN {X 0,Y 496.373,Z 640.586,A -85,B 0,C 180,E1 -6032.841,E2 -6032.841} C_VEL
LIN {X 0,Y 496.901,Z 629.875,A -85,B 0,C 180,E1 -6034.258,E2 -6034.258} C_VEL
LIN {X 0,Y 497.495,Z 618.916,A -85,B 0,C 180,E1 -6035.472,E2 -6035.472} C_VEL
LIN {X 0,Y 498.159,Z 606.922,A -85,B 0,C 180,E1 -6036.582,E2 -6036.582} C_VEL
LIN {X 0,Y 498.787,Z 593.798,A -85,B 0,C 180,E1 -6037.591,E2 -6037.591} C_VEL
LIN {X 0,Y 499.495,Z 579.164,A -85,B 0,C 180,E1 -6038.496,E2 -6038.496} C_VEL
LIN {X 0,Y 500.059,Z 564.683,A -85,B 0,C 180,E1 -6039.199,E2 -6039.199} C_VEL
LIN {X 0,Y 500.538,Z 550.372,A -85,B 0,C 180,E1 -6039.725,E2 -6039.725} C_VEL
LIN {X 0,Y 500.783,Z 535.311,A -85,B 0,C 180,E1 -6040.118,E2 -6040.118} C_VEL
LIN {X 0,Y 501.497,Z 472.471,A -85,B 0,C 180,E1 -6041.059,E2 -6041.059} C_VEL
LIN {X 0,Y 502.109,Z 385.832,A -85,B 0,C 180,E1 -6042.342,E2 -6042.342} C_VEL
LIN {X 0,Y 498.323,Z 369.611,A -85,B 0,C 180,E1 -6042.782,E2 -6042.782} C_VEL
LIN {X 0,Y 498.362,Z 364.358,A -85,B 0,C 180,E1 -6043.638,E2 -6043.638} C_VEL
LIN {X 0,Y 495.793,Z 352.355,A -85,B 0,C 180,E1 -6045.783,E2 -6045.783} C_VEL
LIN {X 0,Y 495.777,Z 352.355,A -85,B 0,C 180,E1 -6049.029,E2 -6049.029} C_VEL
LIN {X 0,Y 495.746,Z 352.359,A -85,B 0,C 180,E1 -6051.629,E2 -6051.629} C_VEL
LIN {X 0,Y 495.718,Z 352.358,A -85,B 0,C 180,E1 -6054.277,E2 -6054.277} C_VEL
LIN {X 0,Y 495.737,Z 352.357,A -85,B 0,C 180,E1 -6056.979,E2 -6056.979} C_VEL
LIN {X 0,Y 495.764,Z 352.352,A -85,B 0,C 180,E1 -6060.146,E2 -6060.146} C_VEL
LIN {X 0,Y 495.795,Z 352.348,A -85,B 0,C 180,E1 -6063.244,E2 -6063.244} C_VEL
LIN {X 0,Y 495.7,Z 352.358,A -85,B 0,C 180,E1 -6066.084,E2 -6066.084} C_VEL
LIN {X 0,Y 495.746,Z 352.354,A -85,B 0,C 180,E1 -6068.765,E2 -6068.765} C_VEL
LIN {X 0,Y 495.727,Z 352.361,A -85,B 0,C 180,E1 -6071.784,E2 -6071.784} C_VEL
LIN {X 0,Y 495.741,Z 352.355,A -85,B 0,C 180,E1 -6075.141,E2 -6075.141} C_VEL
LIN {X 0,Y 495.747,Z 352.354,A -85,B 0,C 180,E1 -6078.217,E2 -6078.217} C_VEL
LIN {X 0,Y 495.744,Z 352.356,A -85,B 0,C 180,E1 -6081.235,E2 -6081.235} C_VEL
LIN {X 0,Y 495.745,Z 352.353,A -85,B 0,C 180,E1 -6084.461,E2 -6084.461} C_VEL
LIN {X 0,Y 495.756,Z 352.357,A -85,B 0,C 180,E1 -6087.404,E2 -6087.404} C_VEL
LIN {X 0,Y 495.766,Z 352.349,A -85,B 0,C 180,E1 -6090.253,E2 -6090.253} C_VEL
LIN {X 0,Y 495.742,Z 352.343,A -85,B 0,C 180,E1 -6093.27,E2 -6093.27} C_VEL
LIN {X 0,Y 495.743,Z 352.348,A -85,B 0,C 180,E1 -6096.612,E2 -6096.612} C_VEL
LIN {X 0,Y 495.783,Z 352.353,A -85,B 0,C 180,E1 -6099.324,E2 -6099.324} C_VEL
LIN {X 0,Y 495.783,Z 352.348,A -85,B 0,C 180,E1 -6101.828,E2 -6101.828} C_VEL
LIN {X 0,Y 495.827,Z 352.342,A -85,B 0,C 180,E1 -6104.548,E2 -6104.548} C_VEL
LIN {X 0,Y 495.832,Z 352.339,A -85,B 0,C 180,E1 -6107.965,E2 -6107.965} C_VEL
LIN {X 0,Y 495.81,Z 352.345,A -85,B 0,C 180,E1 -6111.029,E2 -6111.029} C_VEL
LIN {X 0,Y 495.825,Z 352.349,A -85,B 0,C 180,E1 -6113.489,E2 -6113.489} C_VEL
LIN {X 0,Y 495.712,Z 352.359,A -85,B 0,C 180,E1 -6115.935,E2 -6115.935} C_VEL
LIN {X 0,Y 495.98,Z 352.33,A -85,B 0,C 180,E1 -6117.563,E2 -6117.563} C_VEL
LIN {X 0,Y 495.978,Z 352.324,A -85,B 0,C 180,E1 -6120,E2 -6120} C_VEL
LIN {X 0,Y 495.987,Z 352.32,A -85,B 0,C 180,E1 -6122.436,E2 -6122.436} C_VEL
LIN {X 0,Y 495.859,Z 352.345,A -85,B 0,C 180,E1 -6125.694,E2 -6125.694} C_VEL
LIN {X 0,Y 495.832,Z 352.341,A -85,B 0,C 180,E1 -6128.148,E2 -6128.148} C_VEL
LIN {X 0,Y 495.853,Z 352.346,A -85,B 0,C 180,E1 -6131.445,E2 -6131.445} C_VEL
LIN {X 0,Y 495.781,Z 352.347,A -85,B 0,C 180,E1 -6134.783,E2 -6134.783} C_VEL
LIN {X 0,Y 495.773,Z 352.348,A -85,B 0,C 180,E1 -6138.234,E2 -6138.234} C_VEL
LIN {X 0,Y 495.776,Z 352.348,A -85,B 0,C 180,E1 -6140.756,E2 -6140.756} C_VEL
LIN {X 0,Y 495.74,Z 352.356,A -85,B 0,C 180,E1 -6143.387,E2 -6143.387} C_VEL
LIN {X 0,Y 495.743,Z 352.351,A -85,B 0,C 180,E1 -6146.73,E2 -6146.73} C_VEL
LIN {X 0,Y 495.758,Z 352.357,A -85,B 0,C 180,E1 -6149.747,E2 -6149.747} C_VEL
LIN {X 0,Y 495.768,Z 352.349,A -85,B 0,C 180,E1 -6152.594,E2 -6152.594} C_VEL
LIN {X 0,Y 495.736,Z 352.361,A -85,B 0,C 180,E1 -6155.538,E2 -6155.538} C_VEL
LIN {X 0,Y 495.74,Z 352.352,A -85,B 0,C 180,E1 -6158.764,E2 -6158.764} C_VEL
LIN {X 0,Y 495.725,Z 352.362,A -85,B 0,C 180,E1 -6161.784,E2 -6161.784} C_VEL
LIN {X 0,Y 495.737,Z 352.357,A -85,B 0,C 180,E1 -6165.141,E2 -6165.141} C_VEL
LIN {X 0,Y 495.743,Z 352.357,A -85,B 0,C 180,E1 -6168.217,E2 -6168.217} C_VEL
LIN {X 0,Y 495.74,Z 352.36,A -85,B 0,C 180,E1 -6171.235,E2 -6171.235} C_VEL
LIN {X 0,Y 495.742,Z 352.356,A -85,B 0,C 180,E1 -6174.462,E2 -6174.462} C_VEL
LIN {X 0,Y 495.766,Z 352.358,A -85,B 0,C 180,E1 -6177.405,E2 -6177.405} C_VEL
LIN {X 0,Y 495.81,Z 352.507,A -85,B 0,C 180,E1 -6180.81,E2 -6180.81} C_VEL
LIN {X 0,Y 499.416,Z 368.053,A -85,B 0,C 180,E1 -6183.236,E2 -6183.236} C_VEL
LIN {X 0,Y 499.261,Z 376.396,A -85,B 0,C 180,E1 -6184.406,E2 -6184.406} C_VEL
LIN {X 0,Y 498.373,Z 397.173,A -85,B 0,C 180,E1 -6187.261,E2 -6187.261} C_VEL
LIN {X 0,Y 502.12,Z 417.161,A -85,B 0,C 180,E1 -6187.742,E2 -6187.742} C_VEL
LIN {X 0,Y 500.799,Z 563.239,A -85,B 0,C 180,E1 -6189.903,E2 -6189.903} C_VEL
LIN {X 0,Y 500.34,Z 579.108,A -85,B 0,C 180,E1 -6190.299,E2 -6190.299} C_VEL
LIN {X 0,Y 499.846,Z 594.085,A -85,B 0,C 180,E1 -6190.846,E2 -6190.846} C_VEL
LIN {X 0,Y 499.248,Z 608.342,A -85,B 0,C 180,E1 -6191.534,E2 -6191.534} C_VEL
LIN {X 0,Y 498.621,Z 621.886,A -85,B 0,C 180,E1 -6192.36,E2 -6192.36} C_VEL
LIN {X 0,Y 497.991,Z 634.373,A -85,B 0,C 180,E1 -6193.289,E2 -6193.289} C_VEL
LIN {X 0,Y 497.317,Z 647.071,A -85,B 0,C 180,E1 -6194.425,E2 -6194.425} C_VEL
LIN {X 0,Y 496.74,Z 658.609,A -85,B 0,C 180,E1 -6195.665,E2 -6195.665} C_VEL
LIN {X 0,Y 496.265,Z 668.322,A -85,B 0,C 180,E1 -6196.904,E2 -6196.904} C_VEL
LIN {X 0,Y 495.798,Z 677.752,A -85,B 0,C 180,E1 -6198.328,E2 -6198.328} C_VEL
LIN {X 0,Y 495.502,Z 685.811,A -85,B 0,C 180,E1 -6199.788,E2 -6199.788} C_VEL
LIN {X 0,Y 495.27,Z 693.232,A -85,B 0,C 180,E1 -6201.431,E2 -6201.431} C_VEL
LIN {X 0,Y 495.151,Z 699.121,A -85,B 0,C 180,E1 -6203.071,E2 -6203.071} C_VEL
LIN {X 0,Y 495.076,Z 702.62,A -85,B 0,C 180,E1 -6204.297,E2 -6204.297} C_VEL
LIN {X 0,Y 494.991,Z 706.155,A -85,B 0,C 180,E1 -6205.929,E2 -6205.929} C_VEL
LIN {X 0,Y 494.994,Z 708.482,A -85,B 0,C 180,E1 -6207.559,E2 -6207.559} C_VEL
LIN {X 0,Y 494.907,Z 709.649,A -85,B 0,C 180,E1 -6209.186,E2 -6209.186} C_VEL
LIN {X 0,Y 494.907,Z 709.646,A -85,B 0,C 180,E1 -6210.814,E2 -6210.814} C_VEL
LIN {X 0,Y 494.994,Z 708.472,A -85,B 0,C 180,E1 -6212.441,E2 -6212.441} C_VEL
LIN {X 0,Y 494.991,Z 706.141,A -85,B 0,C 180,E1 -6214.071,E2 -6214.071} C_VEL
LIN {X 0,Y 495.07,Z 702.607,A -85,B 0,C 180,E1 -6215.703,E2 -6215.703} C_VEL
LIN {X 0,Y 495.161,Z 697.778,A -85,B 0,C 180,E1 -6217.339,E2 -6217.339} C_VEL
LIN {X 0,Y 495.31,Z 691.523,A -85,B 0,C 180,E1 -6218.979,E2 -6218.979} C_VEL
LIN {X 0,Y 495.616,Z 683.671,A -85,B 0,C 180,E1 -6220.623,E2 -6220.623} C_VEL
LIN {X 0,Y 495.898,Z 675.277,A -85,B 0,C 180,E1 -6222.072,E2 -6222.072} C_VEL
LIN {X 0,Y 496.411,Z 665.26,A -85,B 0,C 180,E1 -6223.509,E2 -6223.509} C_VEL
LIN {X 0,Y 496.873,Z 654.973,A -85,B 0,C 180,E1 -6224.75,E2 -6224.75} C_VEL
LIN {X 0,Y 497.615,Z 642.138,A -85,B 0,C 180,E1 -6226.04,E2 -6226.04} C_VEL
LIN {X 0,Y 498.208,Z 629.08,A -85,B 0,C 180,E1 -6227.126,E2 -6227.126} C_VEL
LIN {X 0,Y 498.98,Z 615.411,A -85,B 0,C 180,E1 -6228.051,E2 -6228.051} C_VEL
LIN {X 0,Y 499.576,Z 601.25,A -85,B 0,C 180,E1 -6228.825,E2 -6228.825} C_VEL
LIN {X 0,Y 500.077,Z 587.267,A -85,B 0,C 180,E1 -6229.421,E2 -6229.421} C_VEL
LIN {X 0,Y 500.579,Z 571.639,A -85,B 0,C 180,E1 -6229.908,E2 -6229.908} C_VEL
LIN {X 0,Y 500.854,Z 555.634,A -85,B 0,C 180,E1 -6230.227,E2 -6230.227} C_VEL
LIN {X 0,Y 502.057,Z 415.992,A -85,B 0,C 180,E1 -6232.28,E2 -6232.28} C_VEL
LIN {X 0,Y 498.38,Z 397.048,A -85,B 0,C 180,E1 -6232.75,E2 -6232.75} C_VEL
LIN {X 0,Y 499.334,Z 376.485,A -85,B 0,C 180,E1 -6235.597,E2 -6235.597} C_VEL
LIN {X 0,Y 499.479,Z 368.304,A -85,B 0,C 180,E1 -6236.76,E2 -6236.76} C_VEL
LIN {X 0,Y 496.241,Z 354.216,A -85,B 0,C 180,E1 -6239.017,E2 -6239.017} C_VEL
LIN {X 0,Y 495.796,Z 352.35,A -85,B 0,C 180,E1 -6239.336,E2 -6239.336} C_VEL
LIN {X 0,Y 495.765,Z 352.358,A -85,B 0,C 180,E1 -6242.595,E2 -6242.595} C_VEL
LIN {X 0,Y 495.741,Z 352.357,A -85,B 0,C 180,E1 -6245.538,E2 -6245.538} C_VEL
LIN {X 0,Y 495.74,Z 352.355,A -85,B 0,C 180,E1 -6248.765,E2 -6248.765} C_VEL
LIN {X 0,Y 495.742,Z 352.354,A -85,B 0,C 180,E1 -6251.783,E2 -6251.783} C_VEL
LIN {X 0,Y 495.736,Z 352.356,A -85,B 0,C 180,E1 -6255.141,E2 -6255.141} C_VEL
LIN {X 0,Y 495.722,Z 352.362,A -85,B 0,C 180,E1 -6258.216,E2 -6258.216} C_VEL
LIN {X 0,Y 495.74,Z 352.355,A -85,B 0,C 180,E1 -6261.235,E2 -6261.235} C_VEL
LIN {X 0,Y 495.743,Z 352.353,A -85,B 0,C 180,E1 -6264.462,E2 -6264.462} C_VEL
LIN {X 0,Y 495.767,Z 352.349,A -85,B 0,C 180,E1 -6267.406,E2 -6267.406} C_VEL
LIN {X 0,Y 495.762,Z 352.347,A -85,B 0,C 180,E1 -6270.254,E2 -6270.254} C_VEL
LIN {X 0,Y 495.774,Z 352.348,A -85,B 0,C 180,E1 -6273.263,E2 -6273.263} C_VEL
LIN {X 0,Y 495.74,Z 352.357,A -85,B 0,C 180,E1 -6276.613,E2 -6276.613} C_VEL
LIN {X 0,Y 495.78,Z 352.349,A -85,B 0,C 180,E1 -6279.325,E2 -6279.325} C_VEL
LIN {X 0,Y 495.78,Z 352.35,A -85,B 0,C 180,E1 -6281.829,E2 -6281.829} C_VEL
LIN {X 0,Y 495.781,Z 352.349,A -85,B 0,C 180,E1 -6285.217,E2 -6285.217} C_VEL
LIN {X 0,Y 495.852,Z 352.346,A -85,B 0,C 180,E1 -6288.555,E2 -6288.555} C_VEL
LIN {X 0,Y 495.832,Z 352.341,A -85,B 0,C 180,E1 -6291.852,E2 -6291.852} C_VEL
LIN {X 0,Y 495.832,Z 352.34,A -85,B 0,C 180,E1 -6295.122,E2 -6295.122} C_VEL
LIN {X 0,Y 495.988,Z 352.324,A -85,B 0,C 180,E1 -6297.564,E2 -6297.564} C_VEL
LIN {X 0,Y 495.944,Z 352.333,A -85,B 0,C 180,E1 -6300.812,E2 -6300.812} C_VEL
LIN {X 0,Y 495.986,Z 352.33,A -85,B 0,C 180,E1 -6302.437,E2 -6302.437} C_VEL
LIN {X 0,Y 495.874,Z 352.338,A -85,B 0,C 180,E1 -6305.694,E2 -6305.694} C_VEL
LIN {X 0,Y 495.833,Z 352.345,A -85,B 0,C 180,E1 -6308.97,E2 -6308.97} C_VEL
LIN {X 0,Y 495.831,Z 352.343,A -85,B 0,C 180,E1 -6312.035,E2 -6312.035} C_VEL
LIN {X 0,Y 495.827,Z 352.342,A -85,B 0,C 180,E1 -6315.452,E2 -6315.452} C_VEL
LIN {X 0,Y 495.782,Z 352.339,A -85,B 0,C 180,E1 -6319.029,E2 -6319.029} C_VEL
LIN {X 0,Y 495.746,Z 352.351,A -85,B 0,C 180,E1 -6321.629,E2 -6321.629} C_VEL
LIN {X 0,Y 495.718,Z 352.362,A -85,B 0,C 180,E1 -6324.277,E2 -6324.277} C_VEL
LIN {X 0,Y 495.737,Z 352.356,A -85,B 0,C 180,E1 -6326.979,E2 -6326.979} C_VEL
LIN {X 0,Y 495.768,Z 352.353,A -85,B 0,C 180,E1 -6330.147,E2 -6330.147} C_VEL
LIN {X 0,Y 495.793,Z 352.349,A -85,B 0,C 180,E1 -6333.244,E2 -6333.244} C_VEL
LIN {X 0,Y 495.711,Z 352.354,A -85,B 0,C 180,E1 -6336.087,E2 -6336.087} C_VEL
LIN {X 0,Y 495.744,Z 352.354,A -85,B 0,C 180,E1 -6338.765,E2 -6338.765} C_VEL
LIN {X 0,Y 495.747,Z 352.355,A -85,B 0,C 180,E1 -6341.783,E2 -6341.783} C_VEL
LIN {X 0,Y 495.741,Z 352.354,A -85,B 0,C 180,E1 -6345.141,E2 -6345.141} C_VEL
LIN {X 0,Y 495.754,Z 352.355,A -85,B 0,C 180,E1 -6348.218,E2 -6348.218} C_VEL
LIN {X 0,Y 495.752,Z 352.355,A -85,B 0,C 180,E1 -6351.408,E2 -6351.408} C_VEL
LIN {X 0,Y 495.766,Z 352.496,A -85,B 0,C 180,E1 -6354.262,E2 -6354.262} C_VEL
LIN {X 0,Y 498.361,Z 363.759,A -85,B 0,C 180,E1 -6356.309,E2 -6356.309} C_VEL
LIN {X 0,Y 498.405,Z 369.887,A -85,B 0,C 180,E1 -6357.313,E2 -6357.313} C_VEL
LIN {X 0,Y 502.262,Z 386.423,A -85,B 0,C 180,E1 -6357.758,E2 -6357.758} C_VEL
LIN {X 0,Y 502.192,Z 394.914,A -85,B 0,C 180,E1 -6357.884,E2 -6357.884} C_VEL
LIN {X 0,Y 501.587,Z 400.764,A -85,B 0,C 180,E1 -6357.944,E2 -6357.944} C_VEL
LIN {X 0,Y 496.032,Z 419.832,A -85,B 0,C 180,E1 -6357.967,E2 -6357.967} C_VEL
LIN {X 0,Y 495.329,Z 425.689,A -85,B 0,C 180,E1 -6358.024,E2 -6358.024} C_VEL
LIN {X 0,Y 494.172,Z 535.141,A -85,B 0,C 180,E1 -6359.677,E2 -6359.677} C_VEL
LIN {X 0,Y 493.755,Z 550.994,A -85,B 0,C 180,E1 -6360.091,E2 -6360.091} C_VEL
LIN {X 0,Y 493.277,Z 565.572,A -85,B 0,C 180,E1 -6360.641,E2 -6360.641} C_VEL
LIN {X 0,Y 492.668,Z 579.597,A -85,B 0,C 180,E1 -6361.336,E2 -6361.336} C_VEL
LIN {X 0,Y 492.034,Z 594.183,A -85,B 0,C 180,E1 -6362.258,E2 -6362.258} C_VEL
LIN {X 0,Y 491.243,Z 607.876,A -85,B 0,C 180,E1 -6363.329,E2 -6363.329} C_VEL
LIN {X 0,Y 490.579,Z 620.111,A -85,B 0,C 180,E1 -6364.494,E2 -6364.494} C_VEL
LIN {X 0,Y 489.861,Z 632.04,A -85,B 0,C 180,E1 -6365.865,E2 -6365.865} C_VEL
LIN {X 0,Y 489.334,Z 641.647,A -85,B 0,C 180,E1 -6367.183,E2 -6367.183} C_VEL
LIN {X 0,Y 488.844,Z 650.941,A -85,B 0,C 180,E1 -6368.715,E2 -6368.715} C_VEL
LIN {X 0,Y 488.445,Z 658.59,A -85,B 0,C 180,E1 -6370.237,E2 -6370.237} C_VEL
LIN {X 0,Y 488.218,Z 665.064,A -85,B 0,C 180,E1 -6371.822,E2 -6371.822} C_VEL
LIN {X 0,Y 488.066,Z 669.777,A -85,B 0,C 180,E1 -6373.262,E2 -6373.262} C_VEL
LIN {X 0,Y 487.991,Z 674.115,A -85,B 0,C 180,E1 -6374.975,E2 -6374.975} C_VEL
LIN {X 0,Y 487.851,Z 677.126,A -85,B 0,C 180,E1 -6376.674,E2 -6376.674} C_VEL
LIN {X 0,Y 487.932,Z 678.907,A -85,B 0,C 180,E1 -6378.366,E2 -6378.366} C_VEL
LIN {X 0,Y 487.818,Z 679.512,A -85,B 0,C 180,E1 -6380.044,E2 -6380.044} C_VEL
LIN {X 0,Y 487.843,Z 678.91,A -85,B 0,C 180,E1 -6381.717,E2 -6381.717} C_VEL
LIN {X 0,Y 487.979,Z 676.868,A -85,B 0,C 180,E1 -6383.6,E2 -6383.6} C_VEL
LIN {X 0,Y 487.93,Z 674.257,A -85,B 0,C 180,E1 -6385.042,E2 -6385.042} C_VEL
LIN {X 0,Y 488.115,Z 670.13,A -85,B 0,C 180,E1 -6386.698,E2 -6386.698} C_VEL
LIN {X 0,Y 488.152,Z 664.725,A -85,B 0,C 180,E1 -6388.35,E2 -6388.35} C_VEL
LIN {X 0,Y 488.556,Z 657.856,A -85,B 0,C 180,E1 -6390,E2 -6390} C_VEL
LIN {X 0,Y 488.885,Z 649.366,A -85,B 0,C 180,E1 -6391.648,E2 -6391.648} C_VEL
LIN {X 0,Y 489.44,Z 640.364,A -85,B 0,C 180,E1 -6393.087,E2 -6393.087} C_VEL
LIN {X 0,Y 489.905,Z 631.255,A -85,B 0,C 180,E1 -6394.319,E2 -6394.319} C_VEL
LIN {X 0,Y 490.534,Z 620.475,A -85,B 0,C 180,E1 -6395.55,E2 -6395.55} C_VEL
LIN {X 0,Y 491.238,Z 608.73,A -85,B 0,C 180,E1 -6396.675,E2 -6396.675} C_VEL
LIN {X 0,Y 491.854,Z 595.953,A -85,B 0,C 180,E1 -6397.698,E2 -6397.698} C_VEL
LIN {X 0,Y 492.588,Z 583.503,A -85,B 0,C 180,E1 -6398.513,E2 -6398.513} C_VEL
LIN {X 0,Y 493.155,Z 569.078,A -85,B 0,C 180,E1 -6399.278,E2 -6399.278} C_VEL
LIN {X 0,Y 493.723,Z 553.907,A -85,B 0,C 180,E1 -6399.887,E2 -6399.887} C_VEL
LIN {X 0,Y 494.06,Z 538.86,A -85,B 0,C 180,E1 -6400.32,E2 -6400.32} C_VEL
LIN {X 0,Y 494.395,Z 519.99,A -85,B 0,C 180,E1 -6400.65,E2 -6400.65} C_VEL
LIN {X 0,Y 495.579,Z 387.043,A -85,B 0,C 180,E1 -6402.63,E2 -6402.63} C_VEL
LIN {X 0,Y 491.521,Z 369.903,A -85,B 0,C 180,E1 -6403.091,E2 -6403.091} C_VEL
LIN {X 0,Y 491.436,Z 365.52,A -85,B 0,C 180,E1 -6403.82,E2 -6403.82} C_VEL
LIN {X 0,Y 488.754,Z 353.231,A -85,B 0,C 180,E1 -6406.043,E2 -6406.043} C_VEL
LIN {X 0,Y 488.741,Z 353.233,A -85,B 0,C 180,E1 -6409.314,E2 -6409.314} C_VEL
LIN {X 0,Y 488.702,Z 353.236,A -85,B 0,C 180,E1 -6411.957,E2 -6411.957} C_VEL
LIN {X 0,Y 488.704,Z 353.234,A -85,B 0,C 180,E1 -6415.041,E2 -6415.041} C_VEL
LIN {X 0,Y 488.7,Z 353.232,A -85,B 0,C 180,E1 -6418.332,E2 -6418.332} C_VEL
LIN {X 0,Y 488.695,Z 353.235,A -85,B 0,C 180,E1 -6421.18,E2 -6421.18} C_VEL
LIN {X 0,Y 488.728,Z 353.23,A -85,B 0,C 180,E1 -6424.113,E2 -6424.113} C_VEL
LIN {X 0,Y 488.656,Z 353.236,A -85,B 0,C 180,E1 -6427.161,E2 -6427.161} C_VEL
LIN {X 0,Y 488.697,Z 353.226,A -85,B 0,C 180,E1 -6430.341,E2 -6430.341} C_VEL
LIN {X 0,Y 488.677,Z 353.239,A -85,B 0,C 180,E1 -6433.656,E2 -6433.656} C_VEL
LIN {X 0,Y 488.679,Z 353.228,A -85,B 0,C 180,E1 -6436.344,E2 -6436.344} C_VEL
LIN {X 0,Y 488.707,Z 353.236,A -85,B 0,C 180,E1 -6439.673,E2 -6439.673} C_VEL
LIN {X 0,Y 488.664,Z 353.236,A -85,B 0,C 180,E1 -6442.839,E2 -6442.839} C_VEL
LIN {X 0,Y 488.722,Z 353.231,A -85,B 0,C 180,E1 -6445.886,E2 -6445.886} C_VEL
LIN {X 0,Y 488.694,Z 353.233,A -85,B 0,C 180,E1 -6448.82,E2 -6448.82} C_VEL
LIN {X 0,Y 488.701,Z 353.225,A -85,B 0,C 180,E1 -6451.668,E2 -6451.668} C_VEL
LIN {X 0,Y 488.701,Z 353.215,A -85,B 0,C 180,E1 -6454.959,E2 -6454.959} C_VEL
LIN {X 0,Y 488.702,Z 353.233,A -85,B 0,C 180,E1 -6458.043,E2 -6458.043} C_VEL
LIN {X 0,Y 488.743,Z 353.225,A -85,B 0,C 180,E1 -6460.686,E2 -6460.686} C_VEL
LIN {X 0,Y 488.763,Z 353.224,A -85,B 0,C 180,E1 -6464.145,E2 -6464.145} C_VEL
LIN {X 0,Y 488.742,Z 353.228,A -85,B 0,C 180,E1 -6467.543,E2 -6467.543} C_VEL
LIN {X 0,Y 488.758,Z 353.224,A -85,B 0,C 180,E1 -6470.063,E2 -6470.063} C_VEL
LIN {X 0,Y 488.823,Z 353.215,A -85,B 0,C 180,E1 -6472.768,E2 -6472.768} C_VEL
LIN {X 0,Y 488.795,Z 353.215,A -85,B 0,C 180,E1 -6475.051,E2 -6475.051} C_VEL
LIN {X 0,Y 488.946,Z 353.206,A -85,B 0,C 180,E1 -6477.528,E2 -6477.528} C_VEL
LIN {X 0,Y 488.947,Z 353.199,A -85,B 0,C 180,E1 -6480,E2 -6480} C_VEL
LIN {X 0,Y 488.954,Z 353.196,A -85,B 0,C 180,E1 -6482.471,E2 -6482.471} C_VEL
LIN {X 0,Y 488.818,Z 353.22,A -85,B 0,C 180,E1 -6485.776,E2 -6485.776} C_VEL
LIN {X 0,Y 488.781,Z 353.219,A -85,B 0,C 180,E1 -6488.267,E2 -6488.267} C_VEL
LIN {X 0,Y 488.807,Z 353.223,A -85,B 0,C 180,E1 -6491.612,E2 -6491.612} C_VEL
LIN {X 0,Y 488.75,Z 353.224,A -85,B 0,C 180,E1 -6495,E2 -6495} C_VEL
LIN {X 0,Y 488.746,Z 353.222,A -85,B 0,C 180,E1 -6498.442,E2 -6498.442} C_VEL
LIN {X 0,Y 488.708,Z 353.23,A -85,B 0,C 180,E1 -6501.07,E2 -6501.07} C_VEL
LIN {X 0,Y 488.671,Z 353.241,A -85,B 0,C 180,E1 -6503.746,E2 -6503.746} C_VEL
LIN {X 0,Y 488.701,Z 353.229,A -85,B 0,C 180,E1 -6506.922,E2 -6506.922} C_VEL
LIN {X 0,Y 488.719,Z 353.23,A -85,B 0,C 180,E1 -6510.219,E2 -6510.219} C_VEL
LIN {X 0,Y 488.733,Z 353.232,A -85,B 0,C 180,E1 -6513.483,E2 -6513.483} C_VEL
LIN {X 0,Y 488.656,Z 353.237,A -85,B 0,C 180,E1 -6516.35,E2 -6516.35} C_VEL
LIN {X 0,Y 488.687,Z 353.233,A -85,B 0,C 180,E1 -6519.255,E2 -6519.255} C_VEL
LIN {X 0,Y 488.67,Z 353.242,A -85,B 0,C 180,E1 -6521.595,E2 -6521.595} C_VEL
LIN {X 0,Y 488.701,Z 353.231,A -85,B 0,C 180,E1 -6524.802,E2 -6524.802} C_VEL
LIN {X 0,Y 488.666,Z 353.243,A -85,B 0,C 180,E1 -6527.471,E2 -6527.471} C_VEL
LIN {X 0,Y 488.687,Z 353.235,A -85,B 0,C 180,E1 -6530.744,E2 -6530.744} C_VEL
LIN {X 0,Y 488.665,Z 353.241,A -85,B 0,C 180,E1 -6533.867,E2 -6533.867} C_VEL
LIN {X 0,Y 488.735,Z 353.23,A -85,B 0,C 180,E1 -6536.877,E2 -6536.877} C_VEL
LIN {X 0,Y 488.733,Z 353.232,A -85,B 0,C 180,E1 -6540.494,E2 -6540.494} C_VEL
LIN {X 0,Y 492.483,Z 369.313,A -85,B 0,C 180,E1 -6543.058,E2 -6543.058} C_VEL
LIN {X 0,Y 492.576,Z 374.105,A -85,B 0,C 180,E1 -6543.749,E2 -6543.749} C_VEL
LIN {X 0,Y 491.731,Z 393.151,A -85,B 0,C 180,E1 -6546.41,E2 -6546.41} C_VEL
LIN {X 0,Y 491.563,Z 396.954,A -85,B 0,C 180,E1 -6546.937,E2 -6546.937} C_VEL
LIN {X 0,Y 495.522,Z 418.124,A -85,B 0,C 180,E1 -6547.452,E2 -6547.452} C_VEL
LIN {X 0,Y 494.111,Z 563.617,A -85,B 0,C 180,E1 -6549.633,E2 -6549.633} C_VEL
LIN {X 0,Y 493.623,Z 579.541,A -85,B 0,C 180,E1 -6550.043,E2 -6550.043} C_VEL
LIN {X 0,Y 493.082,Z 594.272,A -85,B 0,C 180,E1 -6550.592,E2 -6550.592} C_VEL
LIN {X 0,Y 492.482,Z 608.109,A -85,B 0,C 180,E1 -6551.271,E2 -6551.271} C_VEL
LIN {X 0,Y 491.83,Z 621.656,A -85,B 0,C 180,E1 -6552.108,E2 -6552.108} C_VEL
LIN {X 0,Y 491.113,Z 634.144,A -85,B 0,C 180,E1 -6553.048,E2 -6553.048} C_VEL
LIN {X 0,Y 490.418,Z 646.845,A -85,B 0,C 180,E1 -6554.2,E2 -6554.2} C_VEL
LIN {X 0,Y 489.776,Z 658.384,A -85,B 0,C 180,E1 -6555.456,E2 -6555.456} C_VEL
LIN {X 0,Y 489.274,Z 668.099,A -85,B 0,C 180,E1 -6556.713,E2 -6556.713} C_VEL
LIN {X 0,Y 488.764,Z 677.814,A -85,B 0,C 180,E1 -6558.206,E2 -6558.206} C_VEL
LIN {X 0,Y 488.473,Z 685.59,A -85,B 0,C 180,E1 -6559.639,E2 -6559.639} C_VEL
LIN {X 0,Y 488.186,Z 693.012,A -85,B 0,C 180,E1 -6561.306,E2 -6561.306} C_VEL
LIN {X 0,Y 488.067,Z 698.902,A -85,B 0,C 180,E1 -6562.969,E2 -6562.969} C_VEL
LIN {X 0,Y 487.975,Z 702.4,A -85,B 0,C 180,E1 -6564.214,E2 -6564.214} C_VEL
LIN {X 0,Y 487.89,Z 705.936,A -85,B 0,C 180,E1 -6565.87,E2 -6565.87} C_VEL
LIN {X 0,Y 487.904,Z 708.264,A -85,B 0,C 180,E1 -6567.523,E2 -6567.523} C_VEL
LIN {X 0,Y 487.83,Z 709.431,A -85,B 0,C 180,E1 -6569.174,E2 -6569.174} C_VEL
LIN {X 0,Y 487.83,Z 709.428,A -85,B 0,C 180,E1 -6570.825,E2 -6570.825} C_VEL
LIN {X 0,Y 487.904,Z 708.252,A -85,B 0,C 180,E1 -6572.477,E2 -6572.477} C_VEL
LIN {X 0,Y 487.89,Z 705.919,A -85,B 0,C 180,E1 -6574.13,E2 -6574.13} C_VEL
LIN {X 0,Y 487.969,Z 702.384,A -85,B 0,C 180,E1 -6575.786,E2 -6575.786} C_VEL
LIN {X 0,Y 488.065,Z 697.553,A -85,B 0,C 180,E1 -6577.446,E2 -6577.446} C_VEL
LIN {X 0,Y 488.242,Z 691.296,A -85,B 0,C 180,E1 -6579.111,E2 -6579.111} C_VEL
LIN {X 0,Y 488.593,Z 683.442,A -85,B 0,C 180,E1 -6580.777,E2 -6580.777} C_VEL
LIN {X 0,Y 488.837,Z 675.712,A -85,B 0,C 180,E1 -6582.141,E2 -6582.141} C_VEL
LIN {X 0,Y 489.439,Z 665.026,A -85,B 0,C 180,E1 -6583.705,E2 -6583.705} C_VEL
LIN {X 0,Y 489.934,Z 654.738,A -85,B 0,C 180,E1 -6584.964,E2 -6584.964} C_VEL
LIN {X 0,Y 490.694,Z 642.681,A -85,B 0,C 180,E1 -6586.199,E2 -6586.199} C_VEL
LIN {X 0,Y 491.308,Z 630.185,A -85,B 0,C 180,E1 -6587.267,E2 -6587.267} C_VEL
LIN {X 0,Y 492.109,Z 616.814,A -85,B 0,C 180,E1 -6588.204,E2 -6588.204} C_VEL
LIN {X 0,Y 492.672,Z 604.05,A -85,B 0,C 180,E1 -6588.937,E2 -6588.937} C_VEL
LIN {X 0,Y 493.26,Z 590.03,A -85,B 0,C 180,E1 -6589.577,E2 -6589.577} C_VEL
LIN {X 0,Y 493.768,Z 574.754,A -85,B 0,C 180,E1 -6590.096,E2 -6590.096} C_VEL
LIN {X 0,Y 494.143,Z 559.285,A -85,B 0,C 180,E1 -6590.447,E2 -6590.447} C_VEL
LIN {X 0,Y 495.503,Z 417.07,A -85,B 0,C 180,E1 -6592.578,E2 -6592.578} C_VEL
LIN {X 0,Y 491.587,Z 396.652,A -85,B 0,C 180,E1 -6593.117,E2 -6593.117} C_VEL
LIN {X 0,Y 492.552,Z 377.314,A -85,B 0,C 180,E1 -6595.841,E2 -6595.841} C_VEL
LIN {X 0,Y 492.803,Z 371.364,A -85,B 0,C 180,E1 -6596.694,E2 -6596.694} C_VEL
LIN {X 0,Y 490.613,Z 360.841,A -85,B 0,C 180,E1 -6598.383,E2 -6598.383} C_VEL
LIN {X 0,Y 488.738,Z 353.23,A -85,B 0,C 180,E1 -6599.683,E2 -6599.683} C_VEL
LIN {X 0,Y 488.735,Z 353.231,A -85,B 0,C 180,E1 -6603.123,E2 -6603.123} C_VEL
LIN {X 0,Y 488.664,Z 353.239,A -85,B 0,C 180,E1 -6606.133,E2 -6606.133} C_VEL
LIN {X 0,Y 488.686,Z 353.231,A -85,B 0,C 180,E1 -6609.256,E2 -6609.256} C_VEL
LIN {X 0,Y 488.666,Z 353.239,A -85,B 0,C 180,E1 -6612.528,E2 -6612.528} C_VEL
LIN {X 0,Y 488.7,Z 353.233,A -85,B 0,C 180,E1 -6615.197,E2 -6615.197} C_VEL
LIN {X 0,Y 488.661,Z 353.243,A -85,B 0,C 180,E1 -6618.58,E2 -6618.58} C_VEL
LIN {X 0,Y 488.688,Z 353.235,A -85,B 0,C 180,E1 -6620.95,E2 -6620.95} C_VEL
LIN {X 0,Y 488.665,Z 353.23,A -85,B 0,C 180,E1 -6623.867,E2 -6623.867} C_VEL
LIN {X 0,Y 488.738,Z 353.227,A -85,B 0,C 180,E1 -6626.877,E2 -6626.877} C_VEL
LIN {X 0,Y 488.722,Z 353.218,A -85,B 0,C 180,E1 -6629.781,E2 -6629.781} C_VEL
LIN {X 0,Y 488.724,Z 353.227,A -85,B 0,C 180,E1 -6633.073,E2 -6633.073} C_VEL
LIN {X 0,Y 488.671,Z 353.242,A -85,B 0,C 180,E1 -6636.254,E2 -6636.254} C_VEL
LIN {X 0,Y 488.747,Z 353.226,A -85,B 0,C 180,E1 -6639.176,E2 -6639.176} C_VEL
LIN {X 0,Y 488.747,Z 353.225,A -85,B 0,C 180,E1 -6641.633,E2 -6641.633} C_VEL
LIN {X 0,Y 488.757,Z 353.226,A -85,B 0,C 180,E1 -6645,E2 -6645} C_VEL
LIN {X 0,Y 488.807,Z 353.221,A -85,B 0,C 180,E1 -6648.388,E2 -6648.388} C_VEL
LIN {X 0,Y 488.781,Z 353.219,A -85,B 0,C 180,E1 -6651.733,E2 -6651.733} C_VEL
LIN {X 0,Y 488.83,Z 353.221,A -85,B 0,C 180,E1 -6654.224,E2 -6654.224} C_VEL
LIN {X 0,Y 488.955,Z 353.2,A -85,B 0,C 180,E1 -6657.529,E2 -6657.529} C_VEL
LIN {X 0,Y 488.896,Z 353.211,A -85,B 0,C 180,E1 -6660.824,E2 -6660.824} C_VEL
LIN {X 0,Y 488.953,Z 353.205,A -85,B 0,C 180,E1 -6662.472,E2 -6662.472} C_VEL
LIN {X 0,Y 488.831,Z 353.216,A -85,B 0,C 180,E1 -6665.776,E2 -6665.776} C_VEL
LIN {X 0,Y 488.772,Z 353.224,A -85,B 0,C 180,E1 -6668.268,E2 -6668.268} C_VEL
LIN {X 0,Y 488.808,Z 353.215,A -85,B 0,C 180,E1 -6671.613,E2 -6671.613} C_VEL
LIN {X 0,Y 488.764,Z 353.225,A -85,B 0,C 180,E1 -6675.001,E2 -6675.001} C_VEL
LIN {X 0,Y 488.749,Z 353.223,A -85,B 0,C 180,E1 -6678.443,E2 -6678.443} C_VEL
LIN {X 0,Y 488.71,Z 353.229,A -85,B 0,C 180,E1 -6681.071,E2 -6681.071} C_VEL
LIN {X 0,Y 488.674,Z 353.235,A -85,B 0,C 180,E1 -6683.747,E2 -6683.747} C_VEL
LIN {X 0,Y 488.702,Z 353.233,A -85,B 0,C 180,E1 -6686.922,E2 -6686.922} C_VEL
LIN {X 0,Y 488.727,Z 353.23,A -85,B 0,C 180,E1 -6690.22,E2 -6690.22} C_VEL
LIN {X 0,Y 488.732,Z 353.228,A -85,B 0,C 180,E1 -6693.483,E2 -6693.483} C_VEL
LIN {X 0,Y 488.672,Z 353.234,A -85,B 0,C 180,E1 -6696.353,E2 -6696.353} C_VEL
LIN {X 0,Y 488.691,Z 353.229,A -85,B 0,C 180,E1 -6699.256,E2 -6699.256} C_VEL
LIN {X 0,Y 488.67,Z 353.237,A -85,B 0,C 180,E1 -6702.529,E2 -6702.529} C_VEL
LIN {X 0,Y 488.705,Z 353.23,A -85,B 0,C 180,E1 -6705.198,E2 -6705.198} C_VEL
LIN {X 0,Y 488.696,Z 353.239,A -85,B 0,C 180,E1 -6708.583,E2 -6708.583} C_VEL
LIN {X 0,Y 488.706,Z 353.236,A -85,B 0,C 180,E1 -6710.948,E2 -6710.948} C_VEL
LIN {X 0,Y 488.69,Z 353.269,A -85,B 0,C 180,E1 -6713.933,E2 -6713.933} C_VEL
LIN {X 0,Y 491.551,Z 365.634,A -85,B 0,C 180,E1 -6716.222,E2 -6716.222} C_VEL
LIN {X 0,Y 491.673,Z 370.14,A -85,B 0,C 180,E1 -6716.972,E2 -6716.972} C_VEL
LIN {X 0,Y 495.703,Z 387.445,A -85,B 0,C 180,E1 -6717.45,E2 -6717.45} C_VEL
LIN {X 0,Y 495.329,Z 425.689,A -85,B 0,C 180,E1 -6718.024,E2 -6718.024} C_VEL
LIN {X 0,Y 494.658,Z 431.536,A -85,B 0,C 180,E1 -6718.081,E2 -6718.081} C_VEL
LIN {X 0,Y 489.206,Z 450.604,A -85,B 0,C 180,E1 -6718.11,E2 -6718.11} C_VEL
LIN {X 0,Y 488.475,Z 456.454,A -85,B 0,C 180,E1 -6718.165,E2 -6718.165} C_VEL
LIN {X 0,Y 487.556,Z 535.02,A -85,B 0,C 180,E1 -6719.371,E2 -6719.371} C_VEL
LIN {X 0,Y 487.122,Z 550.988,A -85,B 0,C 180,E1 -6719.79,E2 -6719.79} C_VEL
LIN {X 0,Y 486.624,Z 565.757,A -85,B 0,C 180,E1 -6720.355,E2 -6720.355} C_VEL
LIN {X 0,Y 486.013,Z 579.132,A -85,B 0,C 180,E1 -6721.025,E2 -6721.025} C_VEL
LIN {X 0,Y 485.399,Z 592.141,A -85,B 0,C 180,E1 -6721.841,E2 -6721.841} C_VEL
LIN {X 0,Y 484.631,Z 604.982,A -85,B 0,C 180,E1 -6722.819,E2 -6722.819} C_VEL
LIN {X 0,Y 483.921,Z 617.135,A -85,B 0,C 180,E1 -6723.939,E2 -6723.939} C_VEL
LIN {X 0,Y 483.279,Z 627.363,A -85,B 0,C 180,E1 -6725.056,E2 -6725.056} C_VEL
LIN {X 0,Y 482.638,Z 637.188,A -85,B 0,C 180,E1 -6726.314,E2 -6726.314} C_VEL
LIN {X 0,Y 482.08,Z 646.478,A -85,B 0,C 180,E1 -6727.726,E2 -6727.726} C_VEL
LIN {X 0,Y 481.64,Z 654.866,A -85,B 0,C 180,E1 -6729.258,E2 -6729.258} C_VEL
LIN {X 0,Y 481.28,Z 661.896,A -85,B 0,C 180,E1 -6730.818,E2 -6730.818} C_VEL
LIN {X 0,Y 481.081,Z 668.24,A -85,B 0,C 180,E1 -6732.574,E2 -6732.574} C_VEL
LIN {X 0,Y 480.956,Z 671.959,A -85,B 0,C 180,E1 -6733.881,E2 -6733.881} C_VEL
LIN {X 0,Y 480.838,Z 675.741,A -85,B 0,C 180,E1 -6735.613,E2 -6735.613} C_VEL
LIN {X 0,Y 480.766,Z 678.245,A -85,B 0,C 180,E1 -6737.334,E2 -6737.334} C_VEL
LIN {X 0,Y 480.78,Z 679.526,A -85,B 0,C 180,E1 -6739.045,E2 -6739.045} C_VEL
LIN {X 0,Y 480.725,Z 679.603,A -85,B 0,C 180,E1 -6740.746,E2 -6740.746} C_VEL
LIN {X 0,Y 480.799,Z 678.536,A -85,B 0,C 180,E1 -6742.441,E2 -6742.441} C_VEL
LIN {X 0,Y 480.89,Z 676.323,A -85,B 0,C 180,E1 -6744.128,E2 -6744.128} C_VEL
LIN {X 0,Y 480.948,Z 672.934,A -85,B 0,C 180,E1 -6745.81,E2 -6745.81} C_VEL
LIN {X 0,Y 481.022,Z 668.305,A -85,B 0,C 180,E1 -6747.488,E2 -6747.488} C_VEL
LIN {X 0,Y 481.225,Z 662.317,A -85,B 0,C 180,E1 -6749.163,E2 -6749.163} C_VEL
LIN {X 0,Y 481.565,Z 656.789,A -85,B 0,C 180,E1 -6750.418,E2 -6750.418} C_VEL
LIN {X 0,Y 481.992,Z 648.011,A -85,B 0,C 180,E1 -6752.089,E2 -6752.089} C_VEL
LIN {X 0,Y 482.568,Z 638.695,A -85,B 0,C 180,E1 -6753.549,E2 -6753.549} C_VEL
LIN {X 0,Y 483.16,Z 629.244,A -85,B 0,C 180,E1 -6754.798,E2 -6754.798} C_VEL
LIN {X 0,Y 483.845,Z 618.069,A -85,B 0,C 180,E1 -6756.045,E2 -6756.045} C_VEL
LIN {X 0,Y 484.584,Z 605.823,A -85,B 0,C 180,E1 -6757.186,E2 -6757.186} C_VEL
LIN {X 0,Y 485.264,Z 593.848,A -85,B 0,C 180,E1 -6758.118,E2 -6758.118} C_VEL
LIN {X 0,Y 486.048,Z 579.056,A -85,B 0,C 180,E1 -6759.047,E2 -6759.047} C_VEL
LIN {X 0,Y 486.647,Z 565.601,A -85,B 0,C 180,E1 -6759.717,E2 -6759.717} C_VEL
LIN {X 0,Y 487.147,Z 551.38,A -85,B 0,C 180,E1 -6760.258,E2 -6760.258} C_VEL
LIN {X 0,Y 487.472,Z 536.053,A -85,B 0,C 180,E1 -6760.671,E2 -6760.671} C_VEL
LIN {X 0,Y 488.046,Z 486.491,A -85,B 0,C 180,E1 -6761.442,E2 -6761.442} C_VEL
LIN {X 0,Y 488.977,Z 387.972,A -85,B 0,C 180,E1 -6762.929,E2 -6762.929} C_VEL
LIN {X 0,Y 484.747,Z 369.991,A -85,B 0,C 180,E1 -6763.436,E2 -6763.436} C_VEL
LIN {X 0,Y 484.151,Z 365.113,A -85,B 0,C 180,E1 -6764.287,E2 -6764.287} C_VEL
LIN {X 0,Y 481.691,Z 354.111,A -85,B 0,C 180,E1 -6766.312,E2 -6766.312} C_VEL
LIN {X 0,Y 481.705,Z 354.11,A -85,B 0,C 180,E1 -6769.607,E2 -6769.607} C_VEL
LIN {X 0,Y 481.653,Z 354.112,A -85,B 0,C 180,E1 -6772.295,E2 -6772.295} C_VEL
LIN {X 0,Y 481.673,Z 354.111,A -85,B 0,C 180,E1 -6775.225,E2 -6775.225} C_VEL
LIN {X 0,Y 481.656,Z 354.114,A -85,B 0,C 180,E1 -6777.835,E2 -6777.835} C_VEL
LIN {X 0,Y 481.646,Z 354.11,A -85,B 0,C 180,E1 -6780.711,E2 -6780.711} C_VEL
LIN {X 0,Y 481.702,Z 354.109,A -85,B 0,C 180,E1 -6783.733,E2 -6783.733} C_VEL
LIN {X 0,Y 481.613,Z 354.111,A -85,B 0,C 180,E1 -6786.748,E2 -6786.748} C_VEL
LIN {X 0,Y 481.66,Z 354.106,A -85,B 0,C 180,E1 -6789.942,E2 -6789.942} C_VEL
LIN {X 0,Y 481.623,Z 354.117,A -85,B 0,C 180,E1 -6793.302,E2 -6793.302} C_VEL
LIN {X 0,Y 481.656,Z 354.107,A -85,B 0,C 180,E1 -6795.641,E2 -6795.641} C_VEL
LIN {X 0,Y 481.635,Z 354.112,A -85,B 0,C 180,E1 -6798.955,E2 -6798.955} C_VEL
LIN {X 0,Y 481.638,Z 354.113,A -85,B 0,C 180,E1 -6801.996,E2 -6801.996} C_VEL
LIN {X 0,Y 481.685,Z 354.11,A -85,B 0,C 180,E1 -6805.317,E2 -6805.317} C_VEL
LIN {X 0,Y 481.646,Z 354.111,A -85,B 0,C 180,E1 -6808.311,E2 -6808.311} C_VEL
LIN {X 0,Y 481.668,Z 354.108,A -85,B 0,C 180,E1 -6811.216,E2 -6811.216} C_VEL
LIN {X 0,Y 481.632,Z 354.096,A -85,B 0,C 180,E1 -6814.038,E2 -6814.038} C_VEL
LIN {X 0,Y 481.678,Z 354.1,A -85,B 0,C 180,E1 -6816.812,E2 -6816.812} C_VEL
LIN {X 0,Y 481.699,Z 354.111,A -85,B 0,C 180,E1 -6819.502,E2 -6819.502} C_VEL
LIN {X 0,Y 481.691,Z 354.099,A -85,B 0,C 180,E1 -6822.157,E2 -6822.157} C_VEL
LIN {X 0,Y 481.743,Z 354.097,A -85,B 0,C 180,E1 -6824.775,E2 -6824.775} C_VEL
LIN {X 0,Y 481.754,Z 354.089,A -85,B 0,C 180,E1 -6828.215,E2 -6828.215} C_VEL
LIN {X 0,Y 481.724,Z 354.107,A -85,B 0,C 180,E1 -6831.611,E2 -6831.611} C_VEL
LIN {X 0,Y 481.779,Z 354.088,A -85,B 0,C 180,E1 -6834.139,E2 -6834.139} C_VEL
LIN {X 0,Y 481.912,Z 354.081,A -85,B 0,C 180,E1 -6837.492,E2 -6837.492} C_VEL
LIN {X 0,Y 481.916,Z 354.075,A -85,B 0,C 180,E1 -6840,E2 -6840} C_VEL
LIN {X 0,Y 481.92,Z 354.072,A -85,B 0,C 180,E1 -6842.507,E2 -6842.507} C_VEL
LIN {X 0,Y 481.78,Z 354.096,A -85,B 0,C 180,E1 -6845.861,E2 -6845.861} C_VEL
LIN {X 0,Y 481.737,Z 354.095,A -85,B 0,C 180,E1 -6848.388,E2 -6848.388} C_VEL
LIN {X 0,Y 481.753,Z 354.098,A -85,B 0,C 180,E1 -6851.785,E2 -6851.785} C_VEL
LIN {X 0,Y 481.731,Z 354.1,A -85,B 0,C 180,E1 -6855.224,E2 -6855.224} C_VEL
LIN {X 0,Y 481.707,Z 354.098,A -85,B 0,C 180,E1 -6858.722,E2 -6858.722} C_VEL
LIN {X 0,Y 481.647,Z 354.114,A -85,B 0,C 180,E1 -6861.394,E2 -6861.394} C_VEL
LIN {X 0,Y 481.65,Z 354.111,A -85,B 0,C 180,E1 -6864.114,E2 -6864.114} C_VEL
LIN {X 0,Y 481.674,Z 354.106,A -85,B 0,C 180,E1 -6867.122,E2 -6867.122} C_VEL
LIN {X 0,Y 481.667,Z 354.112,A -85,B 0,C 180,E1 -6869.742,E2 -6869.742} C_VEL
LIN {X 0,Y 481.672,Z 354.105,A -85,B 0,C 180,E1 -6872.674,E2 -6872.674} C_VEL
LIN {X 0,Y 481.622,Z 354.118,A -85,B 0,C 180,E1 -6875.711,E2 -6875.711} C_VEL
LIN {X 0,Y 481.631,Z 354.109,A -85,B 0,C 180,E1 -6878.863,E2 -6878.863} C_VEL
LIN {X 0,Y 481.623,Z 354.117,A -85,B 0,C 180,E1 -6881.908,E2 -6881.908} C_VEL
LIN {X 0,Y 481.653,Z 354.11,A -85,B 0,C 180,E1 -6884.458,E2 -6884.458} C_VEL
LIN {X 0,Y 481.628,Z 354.12,A -85,B 0,C 180,E1 -6887.837,E2 -6887.837} C_VEL
LIN {X 0,Y 481.655,Z 354.114,A -85,B 0,C 180,E1 -6891.139,E2 -6891.139} C_VEL
LIN {X 0,Y 481.657,Z 354.111,A -85,B 0,C 180,E1 -6894.797,E2 -6894.797} C_VEL
LIN {X 0,Y 481.656,Z 354.115,A -85,B 0,C 180,E1 -6897.811,E2 -6897.811} C_VEL
LIN {X 0,Y 481.711,Z 354.312,A -85,B 0,C 180,E1 -6900.261,E2 -6900.261} C_VEL
LIN {X 0,Y 485.546,Z 370.545,A -85,B 0,C 180,E1 -6902.874,E2 -6902.874} C_VEL
LIN {X 0,Y 485.854,Z 373.761,A -85,B 0,C 180,E1 -6903.357,E2 -6903.357} C_VEL
LIN {X 0,Y 484.848,Z 394.422,A -85,B 0,C 180,E1 -6906.281,E2 -6906.281} C_VEL
LIN {X 0,Y 484.764,Z 397.053,A -85,B 0,C 180,E1 -6906.617,E2 -6906.617} C_VEL
LIN {X 0,Y 488.945,Z 419.354,A -85,B 0,C 180,E1 -6907.164,E2 -6907.164} C_VEL
LIN {X 0,Y 487.436,Z 563.081,A -85,B 0,C 180,E1 -6909.341,E2 -6909.341} C_VEL
LIN {X 0,Y 486.922,Z 578.437,A -85,B 0,C 180,E1 -6909.732,E2 -6909.732} C_VEL
LIN {X 0,Y 486.36,Z 594.333,A -85,B 0,C 180,E1 -6910.331,E2 -6910.331} C_VEL
LIN {X 0,Y 485.715,Z 607.815,A -85,B 0,C 180,E1 -6911,E2 -6911} C_VEL
LIN {X 0,Y 485.035,Z 621.398,A -85,B 0,C 180,E1 -6911.849,E2 -6911.849} C_VEL
LIN {X 0,Y 484.267,Z 633.901,A -85,B 0,C 180,E1 -6912.801,E2 -6912.801} C_VEL
LIN {X 0,Y 483.596,Z 645.138,A -85,B 0,C 180,E1 -6913.822,E2 -6913.822} C_VEL
LIN {X 0,Y 482.89,Z 656.364,A -85,B 0,C 180,E1 -6915.029,E2 -6915.029} C_VEL
LIN {X 0,Y 482.389,Z 666.381,A -85,B 0,C 180,E1 -6916.305,E2 -6916.305} C_VEL
LIN {X 0,Y 481.833,Z 675.986,A -85,B 0,C 180,E1 -6917.757,E2 -6917.757} C_VEL
LIN {X 0,Y 481.489,Z 684.354,A -85,B 0,C 180,E1 -6919.274,E2 -6919.274} C_VEL
LIN {X 0,Y 481.185,Z 691.109,A -85,B 0,C 180,E1 -6920.755,E2 -6920.755} C_VEL
LIN {X 0,Y 480.99,Z 697.352,A -85,B 0,C 180,E1 -6922.443,E2 -6922.443} C_VEL
LIN {X 0,Y 480.883,Z 702.182,A -85,B 0,C 180,E1 -6924.128,E2 -6924.128} C_VEL
LIN {X 0,Y 480.794,Z 705.718,A -85,B 0,C 180,E1 -6925.809,E2 -6925.809} C_VEL
LIN {X 0,Y 480.818,Z 708.046,A -85,B 0,C 180,E1 -6927.487,E2 -6927.487} C_VEL
LIN {X 0,Y 480.756,Z 709.213,A -85,B 0,C 180,E1 -6929.162,E2 -6929.162} C_VEL
LIN {X 0,Y 480.756,Z 709.209,A -85,B 0,C 180,E1 -6930.838,E2 -6930.838} C_VEL
LIN {X 0,Y 480.818,Z 708.032,A -85,B 0,C 180,E1 -6932.513,E2 -6932.513} C_VEL
LIN {X 0,Y 480.794,Z 705.698,A -85,B 0,C 180,E1 -6934.191,E2 -6934.191} C_VEL
LIN {X 0,Y 480.874,Z 702.161,A -85,B 0,C 180,E1 -6935.872,E2 -6935.872} C_VEL
LIN {X 0,Y 480.989,Z 697.328,A -85,B 0,C 180,E1 -6937.556,E2 -6937.556} C_VEL
LIN {X 0,Y 481.185,Z 691.07,A -85,B 0,C 180,E1 -6939.245,E2 -6939.245} C_VEL
LIN {X 0,Y 481.575,Z 683.214,A -85,B 0,C 180,E1 -6940.936,E2 -6940.936} C_VEL
LIN {X 0,Y 481.856,Z 675.323,A -85,B 0,C 180,E1 -6942.347,E2 -6942.347} C_VEL
LIN {X 0,Y 482.46,Z 664.793,A -85,B 0,C 180,E1 -6943.908,E2 -6943.908} C_VEL
LIN {X 0,Y 483.003,Z 654.51,A -85,B 0,C 180,E1 -6945.184,E2 -6945.184} C_VEL
LIN {X 0,Y 483.773,Z 643.222,A -85,B 0,C 180,E1 -6946.36,E2 -6946.36} C_VEL
LIN {X 0,Y 484.47,Z 629.985,A -85,B 0,C 180,E1 -6947.518,E2 -6947.518} C_VEL
LIN {X 0,Y 485.305,Z 616.64,A -85,B 0,C 180,E1 -6948.469,E2 -6948.469} C_VEL
LIN {X 0,Y 485.935,Z 603.909,A -85,B 0,C 180,E1 -6949.21,E2 -6949.21} C_VEL
LIN {X 0,Y 486.568,Z 589.531,A -85,B 0,C 180,E1 -6949.875,E2 -6949.875} C_VEL
LIN {X 0,Y 487.118,Z 574.773,A -85,B 0,C 180,E1 -6950.383,E2 -6950.383} C_VEL
LIN {X 0,Y 487.508,Z 559.492,A -85,B 0,C 180,E1 -6950.738,E2 -6950.738} C_VEL
LIN {X 0,Y 489.033,Z 418.366,A -85,B 0,C 180,E1 -6952.882,E2 -6952.882} C_VEL
LIN {X 0,Y 484.816,Z 396.526,A -85,B 0,C 180,E1 -6953.462,E2 -6953.462} C_VEL
LIN {X 0,Y 485.809,Z 377.14,A -85,B 0,C 180,E1 -6956.243,E2 -6956.243} C_VEL
LIN {X 0,Y 485.997,Z 372.874,A -85,B 0,C 180,E1 -6956.866,E2 -6956.866} C_VEL
LIN {X 0,Y 483.237,Z 360.167,A -85,B 0,C 180,E1 -6958.958,E2 -6958.958} C_VEL
LIN {X 0,Y 481.677,Z 354.112,A -85,B 0,C 180,E1 -6960.012,E2 -6960.012} C_VEL
LIN {X 0,Y 481.669,Z 354.114,A -85,B 0,C 180,E1 -6962.674,E2 -6962.674} C_VEL
LIN {X 0,Y 481.628,Z 354.116,A -85,B 0,C 180,E1 -6965.71,E2 -6965.71} C_VEL
LIN {X 0,Y 481.631,Z 354.111,A -85,B 0,C 180,E1 -6968.863,E2 -6968.863} C_VEL
LIN {X 0,Y 481.633,Z 354.111,A -85,B 0,C 180,E1 -6971.911,E2 -6971.911} C_VEL
LIN {X 0,Y 481.653,Z 354.115,A -85,B 0,C 180,E1 -6974.458,E2 -6974.458} C_VEL
LIN {X 0,Y 481.623,Z 354.116,A -85,B 0,C 180,E1 -6977.837,E2 -6977.837} C_VEL
LIN {X 0,Y 481.648,Z 354.115,A -85,B 0,C 180,E1 -6980.656,E2 -6980.656} C_VEL
LIN {X 0,Y 481.617,Z 354.106,A -85,B 0,C 180,E1 -6983.378,E2 -6983.378} C_VEL
LIN {X 0,Y 481.71,Z 354.108,A -85,B 0,C 180,E1 -6986.33,E2 -6986.33} C_VEL
LIN {X 0,Y 481.648,Z 354.098,A -85,B 0,C 180,E1 -6989.418,E2 -6989.418} C_VEL
LIN {X 0,Y 481.667,Z 354.111,A -85,B 0,C 180,E1 -6992.166,E2 -6992.166} C_VEL
LIN {X 0,Y 481.675,Z 354.108,A -85,B 0,C 180,E1 -6994.968,E2 -6994.968} C_VEL
LIN {X 0,Y 481.648,Z 354.108,A -85,B 0,C 180,E1 -6997.705,E2 -6997.705} C_VEL
LIN {X 0,Y 481.701,Z 354.107,A -85,B 0,C 180,E1 -7000.393,E2 -7000.393} C_VEL
LIN {X 0,Y 481.664,Z 354.108,A -85,B 0,C 180,E1 -7003.033,E2 -7003.033} C_VEL
LIN {X 0,Y 481.681,Z 354.106,A -85,B 0,C 180,E1 -7005.639,E2 -7005.639} C_VEL
LIN {X 0,Y 481.752,Z 354.099,A -85,B 0,C 180,E1 -7008.215,E2 -7008.215} C_VEL
LIN {X 0,Y 481.737,Z 354.095,A -85,B 0,C 180,E1 -7011.612,E2 -7011.612} C_VEL
LIN {X 0,Y 481.789,Z 354.097,A -85,B 0,C 180,E1 -7014.14,E2 -7014.14} C_VEL
LIN {X 0,Y 481.921,Z 354.076,A -85,B 0,C 180,E1 -7017.493,E2 -7017.493} C_VEL
LIN {X 0,Y 481.916,Z 354.075,A -85,B 0,C 180,E1 -7020,E2 -7020} C_VEL
LIN {X 0,Y 481.918,Z 354.08,A -85,B 0,C 180,E1 -7022.508,E2 -7022.508} C_VEL
LIN {X 0,Y 481.79,Z 354.094,A -85,B 0,C 180,E1 -7025.861,E2 -7025.861} C_VEL
LIN {X 0,Y 481.731,Z 354.103,A -85,B 0,C 180,E1 -7028.389,E2 -7028.389} C_VEL
LIN {X 0,Y 481.753,Z 354.095,A -85,B 0,C 180,E1 -7031.785,E2 -7031.785} C_VEL
LIN {X 0,Y 481.745,Z 354.097,A -85,B 0,C 180,E1 -7035.225,E2 -7035.225} C_VEL
LIN {X 0,Y 481.71,Z 354.094,A -85,B 0,C 180,E1 -7038.722,E2 -7038.722} C_VEL
LIN {X 0,Y 481.649,Z 354.107,A -85,B 0,C 180,E1 -7041.395,E2 -7041.395} C_VEL
LIN {X 0,Y 481.652,Z 354.112,A -85,B 0,C 180,E1 -7044.115,E2 -7044.115} C_VEL
LIN {X 0,Y 481.677,Z 354.106,A -85,B 0,C 180,E1 -7047.123,E2 -7047.123} C_VEL
LIN {X 0,Y 481.676,Z 354.106,A -85,B 0,C 180,E1 -7049.742,E2 -7049.742} C_VEL
LIN {X 0,Y 481.674,Z 354.113,A -85,B 0,C 180,E1 -7052.675,E2 -7052.675} C_VEL
LIN {X 0,Y 481.632,Z 354.105,A -85,B 0,C 180,E1 -7055.711,E2 -7055.711} C_VEL
LIN {X 0,Y 481.635,Z 354.11,A -85,B 0,C 180,E1 -7058.863,E2 -7058.863} C_VEL
LIN {X 0,Y 481.638,Z 354.113,A -85,B 0,C 180,E1 -7061.911,E2 -7061.911} C_VEL
LIN {X 0,Y 481.657,Z 354.115,A -85,B 0,C 180,E1 -7064.458,E2 -7064.458} C_VEL
LIN {X 0,Y 481.647,Z 354.11,A -85,B 0,C 180,E1 -7067.839,E2 -7067.839} C_VEL
LIN {X 0,Y 481.662,Z 354.115,A -85,B 0,C 180,E1 -7070.655,E2 -7070.655} C_VEL
LIN {X 0,Y 481.638,Z 354.165,A -85,B 0,C 180,E1 -7073.612,E2 -7073.612} C_VEL
LIN {X 0,Y 484.342,Z 365.754,A -85,B 0,C 180,E1 -7075.802,E2 -7075.802} C_VEL
LIN {X 0,Y 484.921,Z 370.356,A -85,B 0,C 180,E1 -7076.613,E2 -7076.613} C_VEL
LIN {X 0,Y 489.234,Z 388.762,A -85,B 0,C 180,E1 -7077.137,E2 -7077.137} C_VEL
LIN {X 0,Y 488.475,Z 456.454,A -85,B 0,C 180,E1 -7078.165,E2 -7078.165} C_VEL
LIN {X 0,Y 487.732,Z 462.303,A -85,B 0,C 180,E1 -7078.22,E2 -7078.22} C_VEL
LIN {X 0,Y 482.239,Z 481.355,A -85,B 0,C 180,E1 -7078.245,E2 -7078.245} C_VEL
LIN {X 0,Y 481.615,Z 487.197,A -85,B 0,C 180,E1 -7078.306,E2 -7078.306} C_VEL
LIN {X 0,Y 480.96,Z 535.12,A -85,B 0,C 180,E1 -7079.058,E2 -7079.058} C_VEL
LIN {X 0,Y 480.507,Z 550.752,A -85,B 0,C 180,E1 -7079.469,E2 -7079.469} C_VEL
LIN {X 0,Y 480.016,Z 565.205,A -85,B 0,C 180,E1 -7080.024,E2 -7080.024} C_VEL
LIN {X 0,Y 479.316,Z 579.797,A -85,B 0,C 180,E1 -7080.761,E2 -7080.761} C_VEL
LIN {X 0,Y 478.561,Z 594.516,A -85,B 0,C 180,E1 -7081.715,E2 -7081.715} C_VEL
LIN {X 0,Y 477.704,Z 607.47,A -85,B 0,C 180,E1 -7082.747,E2 -7082.747} C_VEL
LIN {X 0,Y 476.919,Z 619.962,A -85,B 0,C 180,E1 -7083.96,E2 -7083.96} C_VEL
LIN {X 0,Y 476.075,Z 631.847,A -85,B 0,C 180,E1 -7085.352,E2 -7085.352} C_VEL
LIN {X 0,Y 475.487,Z 641.54,A -85,B 0,C 180,E1 -7086.71,E2 -7086.71} C_VEL
LIN {X 0,Y 474.876,Z 650.922,A -85,B 0,C 180,E1 -7088.285,E2 -7088.285} C_VEL
LIN {X 0,Y 474.432,Z 658.629,A -85,B 0,C 180,E1 -7089.854,E2 -7089.854} C_VEL
LIN {X 0,Y 474.132,Z 665.459,A -85,B 0,C 180,E1 -7091.563,E2 -7091.563} C_VEL
LIN {X 0,Y 473.922,Z 670.599,A -85,B 0,C 180,E1 -7093.191,E2 -7093.191} C_VEL
LIN {X 0,Y 473.85,Z 674.081,A -85,B 0,C 180,E1 -7094.595,E2 -7094.595} C_VEL
LIN {X 0,Y 473.676,Z 677.165,A -85,B 0,C 180,E1 -7096.267,E2 -7096.267} C_VEL
LIN {X 0,Y 473.761,Z 679.315,A -85,B 0,C 180,E1 -7098.261,E2 -7098.261} C_VEL
LIN {X 0,Y 473.654,Z 679.899,A -85,B 0,C 180,E1 -7099.744,E2 -7099.744} C_VEL
LIN {X 0,Y 473.659,Z 679.514,A -85,B 0,C 180,E1 -7101.467,E2 -7101.467} C_VEL
LIN {X 0,Y 473.77,Z 677.986,A -85,B 0,C 180,E1 -7103.184,E2 -7103.184} C_VEL
LIN {X 0,Y 473.784,Z 675.309,A -85,B 0,C 180,E1 -7104.894,E2 -7104.894} C_VEL
LIN {X 0,Y 473.951,Z 671.405,A -85,B 0,C 180,E1 -7106.6,E2 -7106.6} C_VEL
LIN {X 0,Y 474.001,Z 666.21,A -85,B 0,C 180,E1 -7108.301,E2 -7108.301} C_VEL
LIN {X 0,Y 474.422,Z 659.593,A -85,B 0,C 180,E1 -7110,E2 -7110} C_VEL
LIN {X 0,Y 474.823,Z 651.412,A -85,B 0,C 180,E1 -7111.696,E2 -7111.696} C_VEL
LIN {X 0,Y 475.415,Z 642.69,A -85,B 0,C 180,E1 -7113.178,E2 -7113.178} C_VEL
LIN {X 0,Y 476.03,Z 632.276,A -85,B 0,C 180,E1 -7114.658,E2 -7114.658} C_VEL
LIN {X 0,Y 476.732,Z 621.594,A -85,B 0,C 180,E1 -7115.923,E2 -7115.923} C_VEL
LIN {X 0,Y 477.532,Z 609.954,A -85,B 0,C 180,E1 -7117.08,E2 -7117.08} C_VEL
LIN {X 0,Y 478.24,Z 597.303,A -85,B 0,C 180,E1 -7118.132,E2 -7118.132} C_VEL
LIN {X 0,Y 479.107,Z 583.33,A -85,B 0,C 180,E1 -7119.073,E2 -7119.073} C_VEL
LIN {X 0,Y 479.732,Z 569.782,A -85,B 0,C 180,E1 -7119.806,E2 -7119.806} C_VEL
LIN {X 0,Y 480.321,Z 555.412,A -85,B 0,C 180,E1 -7120.406,E2 -7120.406} C_VEL
LIN {X 0,Y 480.712,Z 539.733,A -85,B 0,C 180,E1 -7120.876,E2 -7120.876} C_VEL
LIN {X 0,Y 481.083,Z 520.86,A -85,B 0,C 180,E1 -7121.217,E2 -7121.217} C_VEL
LIN {X 0,Y 482.413,Z 389.308,A -85,B 0,C 180,E1 -7123.225,E2 -7123.225} C_VEL
LIN {X 0,Y 477.883,Z 370.17,A -85,B 0,C 180,E1 -7123.778,E2 -7123.778} C_VEL
LIN {X 0,Y 475.59,Z 359.033,A -85,B 0,C 180,E1 -7125.808,E2 -7125.808} C_VEL
LIN {X 0,Y 474.646,Z 354.988,A -85,B 0,C 180,E1 -7126.588,E2 -7126.588} C_VEL
LIN {X 0,Y 474.657,Z 354.984,A -85,B 0,C 180,E1 -7129.91,E2 -7129.91} C_VEL
LIN {X 0,Y 474.639,Z 354.988,A -85,B 0,C 180,E1 -7133.358,E2 -7133.358} C_VEL
LIN {X 0,Y 474.595,Z 354.989,A -85,B 0,C 180,E1 -7136.376,E2 -7136.376} C_VEL
LIN {X 0,Y 474.605,Z 354.992,A -85,B 0,C 180,E1 -7139.253,E2 -7139.253} C_VEL
LIN {X 0,Y 474.619,Z 354.982,A -85,B 0,C 180,E1 -7142.43,E2 -7142.43} C_VEL
LIN {X 0,Y 474.608,Z 354.991,A -85,B 0,C 180,E1 -7145.467,E2 -7145.467} C_VEL
LIN {X 0,Y 474.594,Z 354.989,A -85,B 0,C 180,E1 -7148.459,E2 -7148.459} C_VEL
LIN {X 0,Y 474.603,Z 354.983,A -85,B 0,C 180,E1 -7150.955,E2 -7150.955} C_VEL
LIN {X 0,Y 474.605,Z 354.987,A -85,B 0,C 180,E1 -7154.106,E2 -7154.106} C_VEL
LIN {X 0,Y 474.579,Z 354.986,A -85,B 0,C 180,E1 -7157.061,E2 -7157.061} C_VEL
LIN {X 0,Y 474.598,Z 354.993,A -85,B 0,C 180,E1 -7159.34,E2 -7159.34} C_VEL
LIN {X 0,Y 474.596,Z 354.993,A -85,B 0,C 180,E1 -7161.707,E2 -7161.707} C_VEL
LIN {X 0,Y 474.622,Z 354.985,A -85,B 0,C 180,E1 -7164.725,E2 -7164.725} C_VEL
LIN {X 0,Y 474.631,Z 354.99,A -85,B 0,C 180,E1 -7167.787,E2 -7167.787} C_VEL
LIN {X 0,Y 474.605,Z 354.985,A -85,B 0,C 180,E1 -7170.889,E2 -7170.889} C_VEL
LIN {X 0,Y 474.585,Z 354.972,A -85,B 0,C 180,E1 -7173.623,E2 -7173.623} C_VEL
LIN {X 0,Y 474.638,Z 354.977,A -85,B 0,C 180,E1 -7176.642,E2 -7176.642} C_VEL
LIN {X 0,Y 474.656,Z 354.982,A -85,B 0,C 180,E1 -7180.089,E2 -7180.089} C_VEL
LIN {X 0,Y 474.638,Z 354.976,A -85,B 0,C 180,E1 -7182.774,E2 -7182.774} C_VEL
LIN {X 0,Y 474.645,Z 354.987,A -85,B 0,C 180,E1 -7185.42,E2 -7185.42} C_VEL
LIN {X 0,Y 474.708,Z 354.968,A -85,B 0,C 180,E1 -7188.037,E2 -7188.037} C_VEL
LIN {X 0,Y 474.699,Z 354.98,A -85,B 0,C 180,E1 -7191.486,E2 -7191.486} C_VEL
LIN {X 0,Y 474.742,Z 354.965,A -85,B 0,C 180,E1 -7194.052,E2 -7194.052} C_VEL
LIN {X 0,Y 474.877,Z 354.957,A -85,B 0,C 180,E1 -7197.455,E2 -7197.455} C_VEL
LIN {X 0,Y 474.885,Z 354.951,A -85,B 0,C 180,E1 -7200,E2 -7200} C_VEL
LIN {X 0,Y 474.886,Z 354.948,A -85,B 0,C 180,E1 -7202.544,E2 -7202.544} C_VEL
LIN {X 0,Y 474.743,Z 354.971,A -85,B 0,C 180,E1 -7205.948,E2 -7205.948} C_VEL
LIN {X 0,Y 474.71,Z 354.97,A -85,B 0,C 180,E1 -7208.513,E2 -7208.513} C_VEL
LIN {X 0,Y 474.706,Z 354.973,A -85,B 0,C 180,E1 -7211.962,E2 -7211.962} C_VEL
LIN {X 0,Y 474.69,Z 354.98,A -85,B 0,C 180,E1 -7215.456,E2 -7215.456} C_VEL
LIN {X 0,Y 474.662,Z 354.977,A -85,B 0,C 180,E1 -7219.01,E2 -7219.01} C_VEL
LIN {X 0,Y 474.589,Z 354.991,A -85,B 0,C 180,E1 -7221.729,E2 -7221.729} C_VEL
LIN {X 0,Y 474.628,Z 354.983,A -85,B 0,C 180,E1 -7224.494,E2 -7224.494} C_VEL
LIN {X 0,Y 474.638,Z 354.985,A -85,B 0,C 180,E1 -7227.324,E2 -7227.324} C_VEL
LIN {X 0,Y 474.598,Z 354.989,A -85,B 0,C 180,E1 -7230.23,E2 -7230.23} C_VEL
LIN {X 0,Y 474.635,Z 354.985,A -85,B 0,C 180,E1 -7233.22,E2 -7233.22} C_VEL
LIN {X 0,Y 474.574,Z 354.991,A -85,B 0,C 180,E1 -7236.325,E2 -7236.325} C_VEL
LIN {X 0,Y 474.6,Z 354.988,A -85,B 0,C 180,E1 -7239.643,E2 -7239.643} C_VEL
LIN {X 0,Y 474.576,Z 354.991,A -85,B 0,C 180,E1 -7242.23,E2 -7242.23} C_VEL
LIN {X 0,Y 474.616,Z 354.99,A -85,B 0,C 180,E1 -7245.298,E2 -7245.298} C_VEL
LIN {X 0,Y 474.603,Z 354.991,A -85,B 0,C 180,E1 -7248.212,E2 -7248.212} C_VEL
LIN {X 0,Y 474.599,Z 354.995,A -85,B 0,C 180,E1 -7251.541,E2 -7251.541} C_VEL
LIN {X 0,Y 474.618,Z 354.987,A -85,B 0,C 180,E1 -7254.725,E2 -7254.725} C_VEL
LIN {X 0,Y 474.634,Z 354.989,A -85,B 0,C 180,E1 -7257.787,E2 -7257.787} C_VEL
LIN {X 0,Y 474.65,Z 355.083,A -85,B 0,C 180,E1 -7259.957,E2 -7259.957} C_VEL
LIN {X 0,Y 478.587,Z 371.804,A -85,B 0,C 180,E1 -7262.691,E2 -7262.691} C_VEL
LIN {X 0,Y 478.952,Z 376.172,A -85,B 0,C 180,E1 -7263.354,E2 -7263.354} C_VEL
LIN {X 0,Y 477.912,Z 396.463,A -85,B 0,C 180,E1 -7266.261,E2 -7266.261} C_VEL
LIN {X 0,Y 482.358,Z 420.444,A -85,B 0,C 180,E1 -7266.87,E2 -7266.87} C_VEL
LIN {X 0,Y 480.751,Z 563.598,A -85,B 0,C 180,E1 -7269.069,E2 -7269.069} C_VEL
LIN {X 0,Y 480.168,Z 579.618,A -85,B 0,C 180,E1 -7269.495,E2 -7269.495} C_VEL
LIN {X 0,Y 479.626,Z 594.24,A -85,B 0,C 180,E1 -7270.06,E2 -7270.06} C_VEL
LIN {X 0,Y 478.874,Z 609.292,A -85,B 0,C 180,E1 -7270.83,E2 -7270.83} C_VEL
LIN {X 0,Y 478.152,Z 622.614,A -85,B 0,C 180,E1 -7271.689,E2 -7271.689} C_VEL
LIN {X 0,Y 477.286,Z 636.143,A -85,B 0,C 180,E1 -7272.762,E2 -7272.762} C_VEL
LIN {X 0,Y 476.483,Z 648.455,A -85,B 0,C 180,E1 -7273.945,E2 -7273.945} C_VEL
LIN {X 0,Y 475.782,Z 659.692,A -85,B 0,C 180,E1 -7275.238,E2 -7275.238} C_VEL
LIN {X 0,Y 475.102,Z 670.587,A -85,B 0,C 180,E1 -7276.745,E2 -7276.745} C_VEL
LIN {X 0,Y 474.614,Z 679.657,A -85,B 0,C 180,E1 -7278.252,E2 -7278.252} C_VEL
LIN {X 0,Y 474.252,Z 687.179,A -85,B 0,C 180,E1 -7279.757,E2 -7279.757} C_VEL
LIN {X 0,Y 474.01,Z 694.198,A -85,B 0,C 180,E1 -7281.473,E2 -7281.473} C_VEL
LIN {X 0,Y 473.887,Z 699.717,A -85,B 0,C 180,E1 -7283.186,E2 -7283.186} C_VEL
LIN {X 0,Y 473.78,Z 703.888,A -85,B 0,C 180,E1 -7284.894,E2 -7284.894} C_VEL
LIN {X 0,Y 473.777,Z 706.813,A -85,B 0,C 180,E1 -7286.598,E2 -7286.598} C_VEL
LIN {X 0,Y 473.721,Z 708.555,A -85,B 0,C 180,E1 -7288.3,E2 -7288.3} C_VEL
LIN {X 0,Y 473.666,Z 709.148,A -85,B 0,C 180,E1 -7290,E2 -7290} C_VEL
LIN {X 0,Y 473.721,Z 708.545,A -85,B 0,C 180,E1 -7291.7,E2 -7291.7} C_VEL
LIN {X 0,Y 473.777,Z 706.793,A -85,B 0,C 180,E1 -7293.402,E2 -7293.402} C_VEL
LIN {X 0,Y 473.778,Z 703.864,A -85,B 0,C 180,E1 -7295.106,E2 -7295.106} C_VEL
LIN {X 0,Y 473.826,Z 699.689,A -85,B 0,C 180,E1 -7296.815,E2 -7296.815} C_VEL
LIN {X 0,Y 474.01,Z 694.161,A -85,B 0,C 180,E1 -7298.526,E2 -7298.526} C_VEL
LIN {X 0,Y 474.252,Z 687.128,A -85,B 0,C 180,E1 -7300.243,E2 -7300.243} C_VEL
LIN {X 0,Y 474.644,Z 679.608,A -85,B 0,C 180,E1 -7301.747,E2 -7301.747} C_VEL
LIN {X 0,Y 475.11,Z 670.546,A -85,B 0,C 180,E1 -7303.255,E2 -7303.255} C_VEL
LIN {X 0,Y 475.774,Z 659.674,A -85,B 0,C 180,E1 -7304.762,E2 -7304.762} C_VEL
LIN {X 0,Y 476.507,Z 648.485,A -85,B 0,C 180,E1 -7306.054,E2 -7306.054} C_VEL
LIN {X 0,Y 477.282,Z 636.247,A -85,B 0,C 180,E1 -7307.238,E2 -7307.238} C_VEL
LIN {X 0,Y 478.142,Z 622.81,A -85,B 0,C 180,E1 -7308.311,E2 -7308.311} C_VEL
LIN {X 0,Y 478.897,Z 609.634,A -85,B 0,C 180,E1 -7309.169,E2 -7309.169} C_VEL
LIN {X 0,Y 479.684,Z 594.812,A -85,B 0,C 180,E1 -7309.939,E2 -7309.939} C_VEL
LIN {X 0,Y 480.302,Z 579.68,A -85,B 0,C 180,E1 -7310.532,E2 -7310.532} C_VEL
LIN {X 0,Y 480.821,Z 564.067,A -85,B 0,C 180,E1 -7310.956,E2 -7310.956} C_VEL
LIN {X 0,Y 481.388,Z 523.497,A -85,B 0,C 180,E1 -7311.603,E2 -7311.603} C_VEL
LIN {X 0,Y 482.434,Z 418.706,A -85,B 0,C 180,E1 -7313.221,E2 -7313.221} C_VEL
LIN {X 0,Y 478.055,Z 396.352,A -85,B 0,C 180,E1 -7313.827,E2 -7313.827} C_VEL
LIN {X 0,Y 479.152,Z 376.737,A -85,B 0,C 180,E1 -7316.693,E2 -7316.693} C_VEL
LIN {X 0,Y 478.92,Z 372.845,A -85,B 0,C 180,E1 -7317.296,E2 -7317.296} C_VEL
LIN {X 0,Y 475.609,Z 358.696,A -85,B 0,C 180,E1 -7319.703,E2 -7319.703} C_VEL
LIN {X 0,Y 474.638,Z 354.989,A -85,B 0,C 180,E1 -7320.374,E2 -7320.374} C_VEL
LIN {X 0,Y 474.624,Z 354.989,A -85,B 0,C 180,E1 -7323.222,E2 -7323.222} C_VEL
LIN {X 0,Y 474.58,Z 354.992,A -85,B 0,C 180,E1 -7326.324,E2 -7326.324} C_VEL
LIN {X 0,Y 474.6,Z 354.987,A -85,B 0,C 180,E1 -7329.644,E2 -7329.644} C_VEL
LIN {X 0,Y 474.587,Z 354.989,A -85,B 0,C 180,E1 -7332.232,E2 -7332.232} C_VEL
LIN {X 0,Y 474.615,Z 354.987,A -85,B 0,C 180,E1 -7335.298,E2 -7335.298} C_VEL
LIN {X 0,Y 474.594,Z 354.994,A -85,B 0,C 180,E1 -7338.212,E2 -7338.212} C_VEL
LIN {X 0,Y 474.617,Z 354.991,A -85,B 0,C 180,E1 -7340.452,E2 -7340.452} C_VEL
LIN {X 0,Y 474.58,Z 354.983,A -85,B 0,C 180,E1 -7343.676,E2 -7343.676} C_VEL
LIN {X 0,Y 474.643,Z 354.984,A -85,B 0,C 180,E1 -7346.78,E2 -7346.78} C_VEL
LIN {X 0,Y 474.601,Z 354.976,A -85,B 0,C 180,E1 -7349.77,E2 -7349.77} C_VEL
LIN {X 0,Y 474.637,Z 354.986,A -85,B 0,C 180,E1 -7352.676,E2 -7352.676} C_VEL
LIN {X 0,Y 474.628,Z 354.985,A -85,B 0,C 180,E1 -7355.506,E2 -7355.506} C_VEL
LIN {X 0,Y 474.635,Z 354.986,A -85,B 0,C 180,E1 -7358.884,E2 -7358.884} C_VEL
LIN {X 0,Y 474.64,Z 354.984,A -85,B 0,C 180,E1 -7361.884,E2 -7361.884} C_VEL
LIN {X 0,Y 474.699,Z 354.979,A -85,B 0,C 180,E1 -7364.545,E2 -7364.545} C_VEL
LIN {X 0,Y 474.706,Z 354.975,A -85,B 0,C 180,E1 -7368.038,E2 -7368.038} C_VEL
LIN {X 0,Y 474.709,Z 354.97,A -85,B 0,C 180,E1 -7371.487,E2 -7371.487} C_VEL
LIN {X 0,Y 474.742,Z 354.969,A -85,B 0,C 180,E1 -7374.904,E2 -7374.904} C_VEL
LIN {X 0,Y 474.886,Z 354.952,A -85,B 0,C 180,E1 -7377.456,E2 -7377.456} C_VEL
LIN {X 0,Y 474.885,Z 354.951,A -85,B 0,C 180,E1 -7380,E2 -7380} C_VEL
LIN {X 0,Y 474.883,Z 354.956,A -85,B 0,C 180,E1 -7382.545,E2 -7382.545} C_VEL
LIN {X 0,Y 474.751,Z 354.971,A -85,B 0,C 180,E1 -7385.948,E2 -7385.948} C_VEL
LIN {X 0,Y 474.706,Z 354.98,A -85,B 0,C 180,E1 -7388.514,E2 -7388.514} C_VEL
LIN {X 0,Y 474.707,Z 354.974,A -85,B 0,C 180,E1 -7391.963,E2 -7391.963} C_VEL
LIN {X 0,Y 474.702,Z 354.974,A -85,B 0,C 180,E1 -7395.456,E2 -7395.456} C_VEL
LIN {X 0,Y 474.665,Z 354.968,A -85,B 0,C 180,E1 -7399.011,E2 -7399.011} C_VEL
LIN {X 0,Y 474.591,Z 354.987,A -85,B 0,C 180,E1 -7401.729,E2 -7401.729} C_VEL
LIN {X 0,Y 474.63,Z 354.982,A -85,B 0,C 180,E1 -7404.495,E2 -7404.495} C_VEL
LIN {X 0,Y 474.64,Z 354.982,A -85,B 0,C 180,E1 -7407.324,E2 -7407.324} C_VEL
LIN {X 0,Y 474.606,Z 354.987,A -85,B 0,C 180,E1 -7410.231,E2 -7410.231} C_VEL
LIN {X 0,Y 474.628,Z 354.986,A -85,B 0,C 180,E1 -7413.222,E2 -7413.222} C_VEL
LIN {X 0,Y 474.584,Z 354.988,A -85,B 0,C 180,E1 -7416.325,E2 -7416.325} C_VEL
LIN {X 0,Y 474.604,Z 354.983,A -85,B 0,C 180,E1 -7419.644,E2 -7419.644} C_VEL
LIN {X 0,Y 474.591,Z 354.991,A -85,B 0,C 180,E1 -7422.232,E2 -7422.232} C_VEL
LIN {X 0,Y 474.62,Z 354.985,A -85,B 0,C 180,E1 -7425.298,E2 -7425.298} C_VEL
LIN {X 0,Y 474.618,Z 354.988,A -85,B 0,C 180,E1 -7428.214,E2 -7428.214} C_VEL
LIN {X 0,Y 474.613,Z 354.989,A -85,B 0,C 180,E1 -7431.543,E2 -7431.543} C_VEL
LIN {X 0,Y 474.601,Z 355.1,A -85,B 0,C 180,E1 -7433.284,E2 -7433.284} C_VEL
LIN {X 0,Y 477.567,Z 367.669,A -85,B 0,C 180,E1 -7435.707,E2 -7435.707} C_VEL
LIN {X 0,Y 478.068,Z 370.46,A -85,B 0,C 180,E1 -7436.222,E2 -7436.222} C_VEL
LIN {X 0,Y 482.725,Z 389.814,A -85,B 0,C 180,E1 -7436.805,E2 -7436.805} C_VEL
LIN {X 0,Y 481.615,Z 487.197,A -85,B 0,C 180,E1 -7438.306,E2 -7438.306} C_VEL
LIN {X 0,Y 480.973,Z 493.046,A -85,B 0,C 180,E1 -7438.367,E2 -7438.367} C_VEL
LIN {X 0,Y 475.374,Z 512.096,A -85,B 0,C 180,E1 -7438.386,E2 -7438.386} C_VEL
LIN {X 0,Y 474.65,Z 517.95,A -85,B 0,C 180,E1 -7438.444,E2 -7438.444} C_VEL
LIN {X 0,Y 474.394,Z 537.733,A -85,B 0,C 180,E1 -7438.793,E2 -7438.793} C_VEL
LIN {X 0,Y 473.873,Z 553.272,A -85,B 0,C 180,E1 -7439.235,E2 -7439.235} C_VEL
LIN {X 0,Y 473.252,Z 568.497,A -85,B 0,C 180,E1 -7439.859,E2 -7439.859} C_VEL
LIN {X 0,Y 472.508,Z 582.391,A -85,B 0,C 180,E1 -7440.604,E2 -7440.604} C_VEL
LIN {X 0,Y 471.754,Z 596.047,A -85,B 0,C 180,E1 -7441.528,E2 -7441.528} C_VEL
LIN {X 0,Y 470.863,Z 608.591,A -85,B 0,C 180,E1 -7442.559,E2 -7442.559} C_VEL
LIN {X 0,Y 470.055,Z 620.829,A -85,B 0,C 180,E1 -7443.779,E2 -7443.779} C_VEL
LIN {X 0,Y 469.162,Z 632.665,A -85,B 0,C 180,E1 -7445.201,E2 -7445.201} C_VEL
LIN {X 0,Y 468.521,Z 642.268,A -85,B 0,C 180,E1 -7446.58,E2 -7446.58} C_VEL
LIN {X 0,Y 467.886,Z 651.46,A -85,B 0,C 180,E1 -7448.16,E2 -7448.16} C_VEL
LIN {X 0,Y 467.388,Z 659.185,A -85,B 0,C 180,E1 -7449.767,E2 -7449.767} C_VEL
LIN {X 0,Y 467.071,Z 666.21,A -85,B 0,C 180,E1 -7451.58,E2 -7451.58} C_VEL
